C05440=1094.394,-80.468,-50.076,175.164,15.276,152.248
C05441=1094.401,-80.195,-50.087,175.166,15.277,152.248
C05442=1094.407,-79.945,-50.099,175.167,15.277,152.247
C05443=1094.413,-79.695,-50.109,175.169,15.278,152.247
C05444=1094.419,-79.446,-50.120,175.170,15.279,152.247
C05445=1094.425,-79.197,-50.131,175.172,15.279,152.247
C05446=1094.431,-78.946,-50.141,175.174,15.280,152.246
C05447=1094.437,-78.696,-50.152,175.175,15.280,152.246
C05448=1094.443,-78.447,-50.163,175.177,15.281,152.246
C05449=1094.448,-78.197,-50.174,175.179,15.282,152.246
C05450=1094.455,-77.947,-50.185,175.181,15.283,152.246
C05451=1094.461,-77.698,-50.195,175.182,15.284,152.245
C05452=1094.467,-77.449,-50.206,175.183,15.284,152.245
C05453=1094.473,-77.199,-50.217,175.185,15.285,152.245
C05454=1094.479,-76.948,-50.228,175.187,15.286,152.245
C05455=1094.484,-76.699,-50.238,175.189,15.286,152.244
C05456=1094.490,-76.449,-50.249,175.191,15.287,152.244
C05457=1094.497,-76.200,-50.260,175.192,15.288,152.244
C05458=1094.503,-75.950,-50.271,175.194,15.288,152.244
C05459=1094.509,-75.700,-50.282,175.195,15.289,152.244
C05460=1094.515,-75.451,-50.293,175.197,15.290,152.243
C05461=1094.521,-75.201,-50.304,175.199,15.291,152.243
C05462=1094.527,-74.951,-50.315,175.201,15.291,152.243
C05463=1094.532,-74.702,-50.326,175.203,15.292,152.243
C05464=1094.539,-74.453,-50.336,175.204,15.292,152.242
C05465=1094.545,-74.202,-50.347,175.205,15.293,152.242
C05466=1094.551,-73.953,-50.358,175.207,15.294,152.242
C05467=1094.557,-73.703,-50.369,175.209,15.295,152.242
C05468=1094.562,-73.453,-50.379,175.211,15.296,152.242
C05469=1094.568,-73.203,-50.390,175.213,15.297,152.241
C05470=1094.574,-72.954,-50.401,175.214,15.297,152.241
C05471=1094.580,-72.704,-50.412,175.215,15.298,152.241
C05472=1094.586,-72.455,-50.423,175.217,15.299,152.241
C05473=1094.592,-72.204,-50.434,175.219,15.299,152.241
C05474=1094.597,-71.955,-50.446,175.221,15.301,152.241
C05475=1094.603,-71.705,-50.457,175.223,15.301,152.240
C05476=1094.608,-71.456,-50.467,175.224,15.302,152.240
C05477=1094.615,-71.205,-50.479,175.225,15.302,152.240
C05478=1094.621,-70.956,-50.490,175.227,15.303,152.240
C05479=1094.627,-70.707,-50.501,175.229,15.304,152.239
C05480=1094.633,-70.457,-50.512,175.231,15.305,152.239
C05481=1094.639,-70.207,-50.523,175.233,15.306,152.239
C05482=1094.644,-69.958,-50.534,175.234,15.306,152.239
C05483=1094.650,-69.708,-50.545,175.236,15.308,152.239
C05484=1094.656,-69.458,-50.556,175.237,15.308,152.238
C05485=1094.662,-69.209,-50.567,175.239,15.308,152.238
C05486=1094.668,-68.959,-50.578,175.241,15.310,152.238
C05487=1094.674,-68.709,-50.589,175.242,15.310,152.238
C05488=1094.680,-68.460,-50.600,175.244,15.311,152.238
C05489=1094.685,-68.210,-50.612,175.246,15.312,152.237
C05490=1094.691,-67.960,-50.623,175.248,15.313,152.237
C05491=1094.697,-67.710,-50.634,175.250,15.314,152.237
C05492=1094.703,-67.461,-50.645,175.250,15.314,152.237
C05493=1094.709,-67.211,-50.657,175.252,15.315,152.237
C05494=1094.715,-66.962,-50.667,175.254,15.316,152.236
C05495=1094.721,-66.712,-50.678,175.256,15.317,152.236
C05496=1094.727,-66.462,-50.690,175.258,15.317,152.236
C05497=1094.733,-66.212,-50.700,175.260,15.318,152.236
C05498=1094.739,-65.963,-50.711,175.261,15.319,152.236
C05499=1094.745,-65.713,-50.724,175.263,15.320,152.235
C05500=1094.750,-65.464,-50.735,175.264,15.321,152.235
C05501=1094.757,-65.213,-50.746,175.266,15.321,152.235
C05502=1094.763,-64.943,-50.758,175.268,15.322,152.235
C05503=1094.769,-64.674,-50.769,175.270,15.323,152.235
C05504=1094.776,-64.404,-50.782,175.272,15.324,152.234
C05505=1094.782,-64.134,-50.794,175.274,15.325,152.234
C05506=1094.788,-63.884,-50.806,175.275,15.325,152.234
C05507=1094.794,-63.634,-50.816,175.277,15.326,152.234
C05508=1094.801,-63.385,-50.828,175.278,15.327,152.234
C05509=1094.806,-63.135,-50.839,175.280,15.328,152.233
C05510=1094.811,-62.885,-50.851,175.282,15.329,152.233
C05511=1094.818,-62.635,-50.862,175.284,15.330,152.233
C05512=1094.824,-62.386,-50.874,175.286,15.330,152.233
C05513=1094.830,-62.136,-50.885,175.287,15.332,152.233
C05514=1094.836,-61.887,-50.896,175.289,15.332,152.232
C05515=1094.842,-61.636,-50.907,175.291,15.333,152.232
C05516=1094.847,-61.387,-50.919,175.292,15.334,152.232
C05517=1094.853,-61.138,-50.930,175.294,15.334,152.232
C05518=1094.860,-60.888,-50.941,175.295,15.335,152.232
C05519=1094.866,-60.639,-50.953,175.297,15.336,152.231
C05520=1094.872,-60.389,-50.964,175.299,15.337,152.231
C05521=1094.878,-60.139,-50.975,175.301,15.338,152.231
C05522=1094.884,-59.889,-50.988,175.303,15.339,152.231
C05523=1094.889,-59.640,-50.998,175.304,15.339,152.230
C05524=1094.896,-59.390,-51.010,175.306,15.341,152.230
C05525=1094.902,-59.141,-51.021,175.308,15.341,152.230
C05526=1094.908,-58.890,-51.032,175.310,15.342,152.230
C05527=1094.913,-58.641,-51.044,175.311,15.343,152.230
C05528=1094.919,-58.392,-51.056,175.312,15.343,152.229
C05529=1094.925,-58.142,-51.067,175.314,15.344,152.229
C05530=1094.931,-57.892,-51.078,175.316,15.345,152.229
C05531=1094.937,-57.642,-51.090,175.318,15.346,152.229
C05532=1094.943,-57.393,-51.101,175.320,15.346,152.229
C05533=1094.949,-57.143,-51.113,175.321,15.348,152.228
C05534=1094.955,-56.894,-51.124,175.323,15.348,152.228
C05535=1094.962,-56.643,-51.135,175.325,15.349,152.228
C05536=1094.967,-56.394,-51.147,175.327,15.350,152.228
C05537=1094.973,-56.144,-51.159,175.329,15.351,152.228
C05538=1094.980,-55.895,-51.171,175.330,15.352,152.227
C05539=1094.986,-55.645,-51.181,175.332,15.353,152.227
C05540=1094.991,-55.395,-51.194,175.334,15.354,152.227
C05541=1094.997,-55.146,-51.205,175.336,15.354,152.227
C05542=1095.004,-54.896,-51.217,175.337,15.355,152.227
C05543=1095.010,-54.647,-51.228,175.339,15.355,152.226
C05544=1095.015,-54.397,-51.240,175.340,15.356,152.226
C05545=1095.021,-54.147,-51.251,175.342,15.357,152.226
C05546=1095.028,-53.898,-51.263,175.344,15.358,152.226
C05547=1095.033,-53.648,-51.275,175.346,15.359,152.225
C05548=1095.040,-53.398,-51.287,175.347,15.360,152.225
C05549=1095.046,-53.148,-51.298,175.349,15.361,152.225
C05550=1095.052,-52.899,-51.309,175.351,15.361,152.225
C05551=1095.058,-52.649,-51.321,175.353,15.363,152.225
C05552=1095.064,-52.400,-51.333,175.355,15.363,152.224
C05553=1095.070,-52.150,-51.344,175.356,15.364,152.224
C05554=1095.076,-51.901,-51.356,175.358,15.365,152.224
C05555=1095.082,-51.650,-51.367,175.360,15.366,152.224
C05556=1095.088,-51.401,-51.379,175.362,15.367,152.224
C05557=1095.094,-51.151,-51.390,175.363,15.368,152.223
C05558=1095.100,-50.901,-51.403,175.365,15.368,152.223
C05559=1095.106,-50.652,-51.414,175.367,15.370,152.223
C05560=1095.112,-50.402,-51.426,175.369,15.370,152.223
C05561=1095.118,-50.153,-51.438,175.371,15.371,152.223
C05562=1095.124,-49.903,-51.449,175.371,15.372,152.223
C05563=1095.129,-49.654,-51.461,175.373,15.372,152.222
C05564=1095.136,-49.404,-51.473,175.375,15.373,152.222
C05565=1095.141,-49.154,-51.485,175.377,15.374,152.222
C05566=1095.147,-48.885,-51.497,175.379,15.376,152.222
C05567=1095.153,-48.616,-51.511,175.381,15.377,152.222
C05568=1095.160,-48.347,-51.523,175.383,15.377,152.221
C05569=1095.166,-48.080,-51.536,175.385,15.378,152.221
C05570=1095.172,-47.829,-51.548,175.386,15.379,152.221
C05571=1095.178,-47.580,-51.559,175.388,15.380,152.221
C05572=1095.184,-47.330,-51.572,175.390,15.381,152.221
C05573=1095.190,-47.080,-51.583,175.392,15.382,152.220
C05574=1095.195,-46.831,-51.595,175.393,15.383,152.220
C05575=1095.202,-46.581,-51.607,175.395,15.384,152.220
C05576=1095.207,-46.332,-51.619,175.397,15.385,152.220
C05577=1095.214,-46.082,-51.631,175.399,15.386,152.220
C05578=1095.219,-45.833,-51.643,175.400,15.387,152.219
C05579=1095.225,-45.583,-51.655,175.402,15.387,152.219
C05580=1095.231,-45.333,-51.667,175.404,15.388,152.219
C05581=1095.237,-45.084,-51.679,175.406,15.389,152.219
C05582=1095.243,-44.834,-51.691,175.408,15.390,152.219
C05583=1095.248,-44.584,-51.702,175.409,15.391,152.218
C05584=1095.255,-44.335,-51.714,175.411,15.392,152.218
C05585=1095.261,-44.085,-51.727,175.413,15.393,152.218
C05586=1095.266,-43.836,-51.739,175.415,15.394,152.218
C05587=1095.272,-43.585,-51.750,175.416,15.394,152.218
C05588=1095.278,-43.335,-51.763,175.418,15.396,152.217
C05589=1095.284,-43.087,-51.774,175.420,15.396,152.217
C05590=1095.290,-42.837,-51.787,175.421,15.398,152.217
C05591=1095.295,-42.587,-51.798,175.423,15.398,152.217
C05592=1095.302,-42.337,-51.810,175.425,15.399,152.217
C05593=1095.308,-42.087,-51.823,175.427,15.400,152.216
C05594=1095.313,-41.838,-51.835,175.429,15.401,152.216
C05595=1095.320,-41.589,-51.847,175.430,15.402,152.216
C05596=1095.326,-41.339,-51.860,175.432,15.403,152.216
C05597=1095.331,-41.089,-51.871,175.434,15.404,152.216
C05598=1095.337,-40.839,-51.883,175.436,15.405,152.216
C05599=1095.343,-40.590,-51.896,175.438,15.405,152.215
C05600=1095.349,-40.341,-51.907,175.439,15.406,152.215
C05601=1095.355,-40.091,-51.920,175.441,15.407,152.215
C05602=1095.361,-39.841,-51.932,175.443,15.408,152.215
C05603=1095.367,-39.591,-51.943,175.445,15.409,152.215
C05604=1095.373,-39.342,-51.956,175.446,15.410,152.214
C05605=1095.379,-39.092,-51.968,175.448,15.411,152.214
C05606=1095.385,-38.842,-51.980,175.450,15.412,152.214
C05607=1095.391,-38.593,-51.992,175.451,15.413,152.214
C05608=1095.397,-38.343,-52.005,175.453,15.414,152.214
C05609=1095.402,-38.094,-52.017,175.455,15.415,152.213
C05610=1095.409,-37.844,-52.029,175.457,15.415,152.213
C05611=1095.414,-37.594,-52.042,175.458,15.417,152.213
C05612=1095.420,-37.345,-52.054,175.460,15.417,152.213
C05613=1095.425,-37.095,-52.066,175.462,15.418,152.213
C05614=1095.431,-36.845,-52.078,175.464,15.419,152.212
C05615=1095.437,-36.596,-52.090,175.466,15.420,152.212
C05616=1095.443,-36.346,-52.102,175.467,15.421,152.212
C05617=1095.449,-36.096,-52.115,175.469,15.422,152.212
C05618=1095.454,-35.847,-52.127,175.471,15.424,152.212
C05619=1095.460,-35.597,-52.140,175.473,15.424,152.211
C05620=1095.467,-35.348,-52.152,175.475,15.425,152.211
C05621=1095.473,-35.098,-52.164,175.477,15.426,152.211
C05622=1095.478,-34.848,-52.176,175.478,15.427,152.211
C05623=1095.484,-34.599,-52.189,175.480,15.428,152.211
C05624=1095.490,-34.349,-52.202,175.482,15.429,152.211
C05625=1095.495,-34.100,-52.214,175.484,15.430,152.210
C05626=1095.501,-33.850,-52.226,175.486,15.431,152.210
C05627=1095.508,-33.600,-52.238,175.487,15.432,152.210
C05628=1095.514,-33.350,-52.251,175.489,15.433,152.210
C05629=1095.519,-33.101,-52.263,175.491,15.434,152.210
C05630=1095.526,-32.832,-52.276,175.493,15.434,152.209
C05631=1095.532,-32.564,-52.290,175.494,15.436,152.209
C05632=1095.538,-32.296,-52.304,175.497,15.437,152.209
C05633=1095.545,-32.028,-52.317,175.499,15.438,152.209
C05634=1095.550,-31.769,-52.330,175.500,15.439,152.209
C05635=1095.557,-31.512,-52.342,175.502,15.439,152.208
C05636=1095.563,-31.253,-52.355,175.504,15.441,152.208
C05637=1095.569,-30.996,-52.369,175.506,15.441,152.208
C05638=1095.575,-30.746,-52.381,175.507,15.443,152.208
C05639=1095.581,-30.497,-52.393,175.510,15.444,152.208
C05640=1095.587,-30.247,-52.406,175.512,15.445,152.207
C05641=1095.593,-29.997,-52.418,175.513,15.446,152.207
C05642=1095.598,-29.747,-52.431,175.515,15.446,152.207
C05643=1095.604,-29.498,-52.443,175.517,15.448,152.207
C05644=1095.610,-29.249,-52.456,175.519,15.448,152.207
C05645=1095.616,-28.999,-52.469,175.521,15.449,152.206
C05646=1095.622,-28.749,-52.481,175.522,15.450,152.206
C05647=1095.628,-28.499,-52.494,175.524,15.451,152.206
C05648=1095.633,-28.250,-52.506,175.526,15.452,152.206
C05649=1095.640,-28.001,-52.519,175.528,15.453,152.206
C05650=1095.646,-27.751,-52.531,175.529,15.454,152.206
C05651=1095.652,-27.501,-52.544,175.531,15.455,152.205
C05652=1095.658,-27.251,-52.556,175.533,15.455,152.205
C05653=1095.664,-27.002,-52.569,175.535,15.457,152.205
C05654=1095.669,-26.753,-52.582,175.537,15.458,152.205
C05655=1095.675,-26.503,-52.594,175.539,15.459,152.205
C05656=1095.681,-26.253,-52.607,175.541,15.460,152.204
C05657=1095.686,-26.003,-52.620,175.542,15.461,152.204
C05658=1095.692,-25.754,-52.633,175.544,15.462,152.204
C05659=1095.698,-25.505,-52.646,175.546,15.463,152.204
C05660=1095.704,-25.255,-52.658,175.548,15.464,152.204
C05661=1095.709,-25.005,-52.671,175.550,15.464,152.203
C05662=1095.716,-24.756,-52.684,175.551,15.465,152.203
C05663=1095.722,-24.506,-52.696,175.553,15.466,152.203
C05664=1095.727,-24.256,-52.709,175.555,15.468,152.203
C05665=1095.733,-24.007,-52.721,175.557,15.469,152.203
C05666=1095.739,-23.757,-52.734,175.559,15.470,152.202
C05667=1095.744,-23.507,-52.748,175.561,15.471,152.202
C05668=1095.750,-23.257,-52.760,175.562,15.472,152.202
C05669=1095.756,-23.008,-52.773,175.564,15.472,152.202
C05670=1095.762,-22.759,-52.786,175.566,15.474,152.202
C05671=1095.768,-22.509,-52.798,175.568,15.474,152.201
C05672=1095.774,-22.260,-52.811,175.570,15.475,152.201
C05673=1095.780,-22.010,-52.824,175.572,15.477,152.201
C05674=1095.786,-21.760,-52.837,175.574,15.477,152.201
C05675=1095.791,-21.510,-52.850,175.575,15.479,152.201
C05676=1095.796,-21.261,-52.863,175.577,15.479,152.200
C05677=1095.803,-21.012,-52.876,175.579,15.481,152.200
C05678=1095.808,-20.762,-52.888,175.581,15.481,152.200
C05679=1095.814,-20.512,-52.901,175.583,15.482,152.200
C05680=1095.821,-20.263,-52.914,175.584,15.483,152.200
C05681=1095.826,-20.013,-52.927,175.586,15.484,152.200
C05682=1095.832,-19.763,-52.941,175.588,15.486,152.199
C05683=1095.838,-19.514,-52.953,175.590,15.486,152.199
C05684=1095.844,-19.264,-52.966,175.592,15.488,152.199
C05685=1095.850,-19.014,-52.979,175.594,15.488,152.199
C05686=1095.855,-18.765,-52.991,175.596,15.489,152.199
C05687=1095.861,-18.516,-53.005,175.597,15.490,152.198
C05688=1095.867,-18.266,-53.018,175.599,15.491,152.198
C05689=1095.873,-18.016,-53.031,175.601,15.492,152.198
C05690=1095.879,-17.767,-53.043,175.603,15.493,152.198
C05691=1095.885,-17.517,-53.057,175.605,15.494,152.197
C05692=1095.890,-17.267,-53.070,175.607,15.495,152.197
C05693=1095.896,-17.018,-53.083,175.609,15.496,152.197
C05694=1095.902,-16.757,-53.097,175.610,15.497,152.197
C05695=1095.909,-16.496,-53.111,175.612,15.498,152.197
C05696=1095.915,-16.235,-53.124,175.614,15.499,152.197
C05697=1095.921,-15.975,-53.138,175.617,15.500,152.196
C05698=1095.927,-15.725,-53.150,175.618,15.501,152.196
C05699=1095.933,-15.476,-53.164,175.620,15.502,152.196
C05700=1095.939,-15.226,-53.176,175.622,15.503,152.196
C05701=1095.944,-14.976,-53.190,175.624,15.504,152.196
C05702=1095.950,-14.726,-53.203,175.625,15.505,152.195
C05703=1095.956,-14.477,-53.216,175.628,15.506,152.195
C05704=1095.961,-14.227,-53.229,175.630,15.507,152.195
C05705=1095.968,-13.977,-53.242,175.631,15.508,152.195
C05706=1095.974,-13.728,-53.256,175.633,15.509,152.195
C05707=1095.979,-13.478,-53.269,175.635,15.510,152.194
C05708=1095.985,-13.229,-53.282,175.637,15.511,152.194
C05709=1095.990,-12.979,-53.295,175.638,15.512,152.194
C05710=1095.997,-12.729,-53.308,175.641,15.513,152.194
C05711=1096.003,-12.480,-53.322,175.643,15.514,152.194
C05712=1096.008,-12.230,-53.335,175.645,15.515,152.193
C05713=1096.014,-11.981,-53.348,175.646,15.516,152.193
C05714=1096.019,-11.732,-53.362,175.648,15.517,152.193
C05715=1096.025,-11.482,-53.374,175.650,15.518,152.193
C05716=1096.031,-11.233,-53.387,175.652,15.519,152.193
C05717=1096.037,-10.983,-53.401,175.654,15.520,152.192
C05718=1096.043,-10.733,-53.414,175.656,15.521,152.192
C05719=1096.048,-10.484,-53.428,175.658,15.522,152.192
C05720=1096.054,-10.234,-53.441,175.660,15.523,152.192
C05721=1096.059,-9.984,-53.454,175.661,15.524,152.192
C05722=1096.066,-9.735,-53.467,175.663,15.525,152.191
C05723=1096.072,-9.486,-53.481,175.666,15.526,152.191
C05724=1096.077,-9.236,-53.495,175.667,15.527,152.191
C05725=1096.083,-8.986,-53.507,175.669,15.528,152.191
C05726=1096.089,-8.737,-53.521,175.671,15.528,152.191
C05727=1096.095,-8.487,-53.534,175.673,15.530,152.190
C05728=1096.100,-8.238,-53.548,175.675,15.530,152.190
C05729=1096.107,-7.987,-53.561,175.677,15.532,152.190
C05730=1096.112,-7.738,-53.575,175.679,15.533,152.190
C05731=1096.119,-7.488,-53.588,175.681,15.534,152.190
C05732=1096.124,-7.239,-53.602,175.682,15.535,152.189
C05733=1096.130,-6.989,-53.615,175.684,15.535,152.189
C05734=1096.136,-6.739,-53.628,175.686,15.536,152.189
C05735=1096.142,-6.490,-53.642,175.688,15.538,152.189
C05736=1096.147,-6.240,-53.656,175.690,15.539,152.189
C05737=1096.153,-5.991,-53.669,175.692,15.539,152.188
C05738=1096.159,-5.742,-53.683,175.694,15.541,152.188
C05739=1096.165,-5.492,-53.695,175.696,15.541,152.188
C05740=1096.170,-5.242,-53.709,175.698,15.542,152.188
C05741=1096.176,-4.993,-53.722,175.700,15.544,152.188
C05742=1096.182,-4.743,-53.736,175.702,15.544,152.187
C05743=1096.188,-4.494,-53.750,175.704,15.545,152.187
C05744=1096.194,-4.244,-53.764,175.705,15.546,152.187
C05745=1096.200,-3.994,-53.777,175.707,15.547,152.187
C05746=1096.206,-3.745,-53.791,175.709,15.548,152.186
C05747=1096.212,-3.495,-53.803,175.711,15.549,152.186
C05748=1096.217,-3.245,-53.817,175.713,15.550,152.186
C05749=1096.224,-2.996,-53.831,175.715,15.551,152.186
C05750=1096.229,-2.747,-53.844,175.717,15.552,152.186
C05751=1096.234,-2.497,-53.858,175.719,15.553,152.185
C05752=1096.240,-2.247,-53.872,175.721,15.555,152.185
C05753=1096.246,-1.998,-53.885,175.723,15.555,152.185
C05754=1096.252,-1.749,-53.899,175.725,15.556,152.185
C05755=1096.257,-1.499,-53.913,175.726,15.557,152.185
C05756=1096.263,-1.250,-53.926,175.728,15.558,152.184
C05757=1096.269,-1.000,-53.940,175.731,15.560,152.184
C05758=1096.275,-0.729,-53.955,175.732,15.560,152.184
C05759=1096.281,-0.458,-53.970,175.734,15.561,152.184
C05760=1096.288,-0.188,-53.985,175.737,15.563,152.184
C05761=1096.294,0.084,-54.000,175.739,15.564,152.183
C05762=1096.299,0.333,-54.013,175.741,15.564,152.183
C05763=1096.305,0.583,-54.027,175.743,15.566,152.183
C05764=1096.312,0.833,-54.041,175.745,15.567,152.183
C05765=1096.317,1.082,-54.055,175.747,15.568,152.182
C05766=1096.322,1.332,-54.069,175.748,15.569,152.182
C05767=1096.328,1.581,-54.082,175.750,15.569,152.182
C05768=1096.333,1.831,-54.096,175.753,15.571,152.182
C05769=1096.340,2.080,-54.110,175.754,15.572,152.182
C05770=1096.345,2.329,-54.124,175.756,15.573,152.181
C05771=1096.351,2.579,-54.138,175.758,15.573,152.181
C05772=1096.357,2.829,-54.152,175.760,15.574,152.181
C05773=1096.363,3.078,-54.166,175.762,15.576,152.181
C05774=1096.369,3.328,-54.179,175.764,15.577,152.181
C05775=1096.374,3.577,-54.193,175.766,15.578,152.181
C05776=1096.380,3.827,-54.207,175.768,15.578,152.180
C05777=1096.385,4.077,-54.221,175.770,15.579,152.180
C05778=1096.391,4.326,-54.234,175.772,15.580,152.180
C05779=1096.398,4.576,-54.249,175.774,15.582,152.180
C05780=1096.403,4.825,-54.263,175.776,15.582,152.179
C05781=1096.409,5.075,-54.277,175.778,15.583,152.179
C05782=1096.414,5.324,-54.291,175.780,15.585,152.179
C05783=1096.420,5.574,-54.304,175.782,15.586,152.179
C05784=1096.426,5.824,-54.318,175.784,15.586,152.178
C05785=1096.432,6.073,-54.333,175.786,15.587,152.178
C05786=1096.438,6.322,-54.347,175.787,15.588,152.178
C05787=1096.443,6.572,-54.361,175.790,15.589,152.178
C05788=1096.449,6.821,-54.374,175.792,15.590,152.178
C05789=1096.455,7.071,-54.388,175.793,15.591,152.177
C05790=1096.461,7.320,-54.403,175.795,15.592,152.177
C05791=1096.467,7.570,-54.417,175.798,15.593,152.177
C05792=1096.472,7.820,-54.430,175.800,15.594,152.177
C05793=1096.478,8.070,-54.445,175.801,15.595,152.177
C05794=1096.484,8.319,-54.459,175.803,15.596,152.176
C05795=1096.489,8.568,-54.473,175.805,15.597,152.176
C05796=1096.496,8.818,-54.486,175.808,15.598,152.176
C05797=1096.502,9.068,-54.501,175.810,15.599,152.176
C05798=1096.508,9.317,-54.515,175.811,15.600,152.175
C05799=1096.513,9.566,-54.529,175.813,15.601,152.175
C05800=1096.519,9.816,-54.543,175.816,15.602,152.175
C05801=1096.525,10.066,-54.558,175.818,15.603,152.175
C05802=1096.530,10.315,-54.572,175.819,15.604,152.175
C05803=1096.536,10.565,-54.586,175.821,15.604,152.174
C05804=1096.542,10.814,-54.600,175.824,15.606,152.174
C05805=1096.548,11.064,-54.614,175.826,15.606,152.174
C05806=1096.554,11.313,-54.628,175.828,15.607,152.173
C05807=1096.560,11.562,-54.642,175.829,15.608,152.173
C05808=1096.566,11.813,-54.656,175.832,15.610,152.173
C05809=1096.571,12.062,-54.670,175.834,15.610,152.173
C05810=1096.577,12.311,-54.685,175.836,15.611,152.173
C05811=1096.583,12.561,-54.699,175.838,15.612,152.172
C05812=1096.589,12.810,-54.714,175.840,15.613,152.172
C05813=1096.594,13.060,-54.728,175.842,15.614,152.172
C05814=1096.600,13.310,-54.742,175.844,15.615,152.172
C05815=1096.606,13.559,-54.756,175.846,15.616,152.171
C05816=1096.612,13.809,-54.770,175.848,15.616,152.171
C05817=1096.618,14.058,-54.785,175.850,15.618,152.171
C05818=1096.624,14.308,-54.798,175.852,15.618,152.171
C05819=1096.629,14.557,-54.814,175.854,15.619,152.170
C05820=1096.635,14.807,-54.828,175.856,15.620,152.170
C05821=1096.641,15.056,-54.842,175.858,15.622,152.170
C05822=1096.648,15.329,-54.858,175.860,15.622,152.170
C05823=1096.654,15.601,-54.873,175.863,15.624,152.169
C05824=1096.660,15.874,-54.889,175.865,15.624,152.169
C05825=1096.667,16.147,-54.905,175.867,15.626,152.169
C05826=1096.672,16.397,-54.919,175.869,15.627,152.169
C05827=1096.678,16.646,-54.934,175.871,15.628,152.169
C05828=1096.684,16.896,-54.948,175.873,15.628,152.168
C05829=1096.689,17.145,-54.963,175.875,15.630,152.168
C05830=1096.695,17.395,-54.977,175.877,15.630,152.168
C05831=1096.701,17.645,-54.992,175.879,15.631,152.167
C05832=1096.706,17.894,-55.006,175.881,15.632,152.167
C05833=1096.712,18.143,-55.020,175.883,15.634,152.167
C05834=1096.718,18.393,-55.035,175.885,15.634,152.167
C05835=1096.724,18.642,-55.049,175.887,15.635,152.167
C05836=1096.730,18.891,-55.064,175.890,15.636,152.166
C05837=1096.735,19.142,-55.079,175.892,15.637,152.166
C05838=1096.741,19.391,-55.093,175.894,15.638,152.166
C05839=1096.747,19.641,-55.107,175.896,15.638,152.166
C05840=1096.753,19.890,-55.122,175.898,15.640,152.165
C05841=1096.759,20.139,-55.136,175.900,15.641,152.165
C05842=1096.765,20.389,-55.151,175.902,15.642,152.165
C05843=1096.770,20.639,-55.166,175.904,15.642,152.165
C05844=1096.776,20.888,-55.180,175.906,15.644,152.164
C05845=1096.782,21.138,-55.195,175.908,15.644,152.164
C05846=1096.787,21.387,-55.209,175.910,15.645,152.164
C05847=1096.793,21.637,-55.225,175.913,15.646,152.164
C05848=1096.799,21.886,-55.239,175.914,15.648,152.163
C05849=1096.804,22.135,-55.253,175.916,15.648,152.163
C05850=1096.811,22.385,-55.268,175.918,15.649,152.163
C05851=1096.815,22.635,-55.283,175.921,15.650,152.163
C05852=1096.822,22.885,-55.298,175.923,15.651,152.162
C05853=1096.828,23.134,-55.312,175.925,15.652,152.162
C05854=1096.832,23.383,-55.327,175.927,15.653,152.162
C05855=1096.839,23.633,-55.342,175.929,15.654,152.162
C05856=1096.844,23.882,-55.356,175.931,15.654,152.161
C05857=1096.851,24.132,-55.371,175.933,15.655,152.161
C05858=1096.856,24.382,-55.386,175.936,15.656,152.161
C05859=1096.862,24.631,-55.401,175.937,15.658,152.161
C05860=1096.868,24.880,-55.415,175.939,15.658,152.161
C05861=1096.873,25.130,-55.431,175.942,15.660,152.160
C05862=1096.879,25.379,-55.445,175.944,15.660,152.160
C05863=1096.885,25.629,-55.459,175.945,15.661,152.160
C05864=1096.890,25.879,-55.475,175.947,15.662,152.159
C05865=1096.896,26.128,-55.489,175.950,15.663,152.159
C05866=1096.902,26.377,-55.504,175.952,15.664,152.159
C05867=1096.908,26.627,-55.519,175.954,15.665,152.159
C05868=1096.914,26.876,-55.534,175.956,15.666,152.158
C05869=1096.919,27.126,-55.548,175.958,15.667,152.158
C05870=1096.925,27.376,-55.564,175.960,15.667,152.158
C05871=1096.931,27.625,-55.578,175.963,15.669,152.158
C05872=1096.937,27.874,-55.593,175.965,15.669,152.157
C05873=1096.942,28.124,-55.608,175.967,15.670,152.157
C05874=1096.949,28.373,-55.623,175.969,15.671,152.157
C05875=1096.954,28.622,-55.638,175.971,15.672,152.157
C05876=1096.960,28.872,-55.653,175.973,15.673,152.156
C05877=1096.966,29.122,-55.667,175.975,15.673,152.156
C05878=1096.971,29.372,-55.683,175.978,15.675,152.156
C05879=1096.977,29.621,-55.697,175.980,15.676,152.155
C05880=1096.983,29.871,-55.713,175.981,15.676,152.155
C05881=1096.988,30.120,-55.728,175.984,15.678,152.155
C05882=1096.994,30.370,-55.743,175.986,15.678,152.155
C05883=1097.000,30.619,-55.758,175.988,15.679,152.154
C05884=1097.005,30.868,-55.773,175.991,15.680,152.154
C05885=1097.011,31.117,-55.788,175.992,15.681,152.154
C05886=1097.017,31.392,-55.805,175.994,15.682,152.154
C05887=1097.023,31.666,-55.821,175.997,15.683,152.153
C05888=1097.030,31.940,-55.838,176.000,15.684,152.153
C05889=1097.037,32.214,-55.854,176.002,15.685,152.153
C05890=1097.042,32.464,-55.870,176.003,15.686,152.153
C05891=1097.048,32.713,-55.884,176.006,15.687,152.152
C05892=1097.054,32.963,-55.900,176.008,15.688,152.152
C05893=1097.059,33.212,-55.915,176.010,15.688,152.152
C05894=1097.065,33.462,-55.930,176.013,15.689,152.151
C05895=1097.070,33.711,-55.945,176.015,15.690,152.151
C05896=1097.076,33.961,-55.960,176.017,15.691,152.151
C05897=1097.082,34.211,-55.975,176.019,15.692,152.151
C05898=1097.088,34.460,-55.990,176.021,15.693,152.150
C05899=1097.094,34.709,-56.006,176.023,15.694,152.150
C05900=1097.100,34.958,-56.021,176.026,15.695,152.150
C05901=1097.105,35.208,-56.036,176.028,15.696,152.150
C05902=1097.111,35.457,-56.051,176.030,15.696,152.149
C05903=1097.117,35.707,-56.067,176.032,15.698,152.149
C05904=1097.122,35.957,-56.082,176.034,15.698,152.149
C05905=1097.128,36.206,-56.097,176.036,15.699,152.148
C05906=1097.134,36.456,-56.112,176.039,15.700,152.148
C05907=1097.140,36.704,-56.128,176.041,15.701,152.148
C05908=1097.145,36.954,-56.143,176.043,15.701,152.148
C05909=1097.151,37.204,-56.159,176.045,15.703,152.147
C05910=1097.157,37.453,-56.173,176.047,15.703,152.147
C05911=1097.163,37.703,-56.189,176.049,15.704,152.147
C05912=1097.169,37.952,-56.204,176.052,15.705,152.146
C05913=1097.174,38.201,-56.220,176.054,15.706,152.146
C05914=1097.180,38.451,-56.235,176.056,15.706,152.146
C05915=1097.185,38.701,-56.250,176.059,15.708,152.146
C05916=1097.191,38.950,-56.265,176.060,15.708,152.145
C05917=1097.197,39.200,-56.281,176.062,15.709,152.145
C05918=1097.202,39.449,-56.297,176.065,15.710,152.145
C05919=1097.209,39.699,-56.312,176.067,15.711,152.144
C05920=1097.214,39.948,-56.327,176.069,15.712,152.144
C05921=1097.220,40.197,-56.343,176.072,15.713,152.144
C05922=1097.225,40.447,-56.359,176.074,15.713,152.144
C05923=1097.231,40.696,-56.373,176.076,15.714,152.143
C05924=1097.237,40.945,-56.389,176.078,15.715,152.143
C05925=1097.243,41.195,-56.405,176.080,15.716,152.143
C05926=1097.248,41.445,-56.420,176.083,15.717,152.142
C05927=1097.253,41.695,-56.436,176.085,15.718,152.142
C05928=1097.260,41.943,-56.451,176.087,15.718,152.142
C05929=1097.265,42.193,-56.467,176.090,15.720,152.142
C05930=1097.271,42.442,-56.483,176.091,15.720,152.141
C05931=1097.276,42.692,-56.498,176.093,15.721,152.141
C05932=1097.283,42.941,-56.513,176.096,15.722,152.141
C05933=1097.288,43.191,-56.529,176.098,15.723,152.140
C05934=1097.294,43.441,-56.545,176.100,15.723,152.140
C05935=1097.299,43.690,-56.560,176.103,15.725,152.140
C05936=1097.305,43.939,-56.576,176.105,15.725,152.140
C05937=1097.311,44.189,-56.592,176.107,15.726,152.139
C05938=1097.316,44.438,-56.608,176.109,15.727,152.139
C05939=1097.322,44.688,-56.623,176.111,15.728,152.139
C05940=1097.327,44.937,-56.638,176.114,15.729,152.138
C05941=1097.334,45.186,-56.654,176.116,15.730,152.138
C05942=1097.339,45.436,-56.669,176.118,15.730,152.138
C05943=1097.345,45.685,-56.685,176.121,15.731,152.137
C05944=1097.350,45.935,-56.701,176.123,15.732,152.137
C05945=1097.356,46.184,-56.717,176.125,15.733,152.137
C05946=1097.361,46.433,-56.732,176.127,15.734,152.137
C05947=1097.367,46.683,-56.749,176.129,15.735,152.136
C05948=1097.373,46.933,-56.764,176.132,15.736,152.136
C05949=1097.378,47.181,-56.780,176.134,15.736,152.136
C05950=1097.384,47.456,-56.798,176.137,15.738,152.135
C05951=1097.390,47.730,-56.815,176.139,15.738,152.135
C05952=1097.397,48.005,-56.832,176.141,15.739,152.135
C05953=1097.403,48.279,-56.850,176.143,15.740,152.134
C05954=1097.408,48.528,-56.865,176.146,15.741,152.134
C05955=1097.414,48.778,-56.882,176.148,15.741,152.134
C05956=1097.420,49.028,-56.897,176.151,15.743,152.133
C05957=1097.426,49.277,-56.913,176.153,15.743,152.133
C05958=1097.431,49.526,-56.929,176.155,15.744,152.133
C05959=1097.437,49.776,-56.945,176.158,15.745,152.132
C05960=1097.442,50.025,-56.961,176.159,15.746,152.132
C05961=1097.448,50.275,-56.977,176.162,15.746,152.132
C05962=1097.453,50.524,-56.993,176.164,15.747,152.132
C05963=1097.459,50.773,-57.008,176.166,15.748,152.131
C05964=1097.465,51.023,-57.024,176.169,15.749,152.131
C05965=1097.471,51.272,-57.041,176.171,15.750,152.131
C05966=1097.476,51.521,-57.056,176.173,15.750,152.130
C05967=1097.482,51.771,-57.072,176.176,15.751,152.130
C05968=1097.488,52.020,-57.088,176.178,15.752,152.130
C05969=1097.494,52.270,-57.104,176.181,15.753,152.129
C05970=1097.500,52.519,-57.120,176.183,15.753,152.129
C05971=1097.505,52.768,-57.136,176.185,15.754,152.129
C05972=1097.511,53.018,-57.152,176.188,15.755,152.128
C05973=1097.517,53.267,-57.168,176.189,15.756,152.128
C05974=1097.522,53.517,-57.185,176.192,15.757,152.128
C05975=1097.528,53.766,-57.201,176.194,15.757,152.127
C05976=1097.533,54.016,-57.216,176.196,15.758,152.127
C05977=1097.539,54.265,-57.232,176.199,15.759,152.127
C05978=1097.545,54.514,-57.249,176.201,15.760,152.126
C05979=1097.551,54.764,-57.265,176.203,15.760,152.126
C05980=1097.556,55.014,-57.280,176.206,15.761,152.126
C05981=1097.562,55.263,-57.297,176.208,15.762,152.125
C05982=1097.568,55.512,-57.313,176.211,15.763,152.125
C05983=1097.573,55.761,-57.329,176.213,15.763,152.125
C05984=1097.579,56.011,-57.346,176.215,15.764,152.124
C05985=1097.584,56.261,-57.361,176.218,15.765,152.124
C05986=1097.590,56.510,-57.377,176.220,15.765,152.124
C05987=1097.596,56.759,-57.394,176.222,15.767,152.123
C05988=1097.602,57.009,-57.410,176.225,15.767,152.123
C05989=1097.608,57.258,-57.426,176.226,15.768,152.123
C05990=1097.614,57.507,-57.442,176.229,15.768,152.122
C05991=1097.619,57.756,-57.459,176.231,15.769,152.122
C05992=1097.624,58.006,-57.474,176.234,15.770,152.122
C05993=1097.630,58.256,-57.491,176.236,15.771,152.121
C05994=1097.636,58.505,-57.507,176.238,15.771,152.121
C05995=1097.642,58.754,-57.523,176.241,15.772,152.121
C05996=1097.648,59.004,-57.539,176.243,15.772,152.120
C05997=1097.653,59.253,-57.556,176.246,15.774,152.120
C05998=1097.659,59.503,-57.573,176.248,15.774,152.120
C05999=1097.665,59.752,-57.589,176.251,15.775,152.119
C06000=1097.671,60.001,-57.605,176.253,15.776,152.119
C06001=1097.677,60.251,-57.621,176.255,15.776,152.118
C06002=1097.683,60.500,-57.638,176.258,15.777,152.118
C06003=1097.688,60.750,-57.654,176.260,15.777,152.118
C06004=1097.694,60.999,-57.671,176.263,15.779,152.117
C06005=1097.700,61.249,-57.687,176.265,15.779,152.117
C06006=1097.706,61.498,-57.703,176.267,15.779,152.117
C06007=1097.711,61.748,-57.720,176.270,15.781,152.116
C06008=1097.717,61.997,-57.736,176.272,15.781,152.116
C06009=1097.723,62.246,-57.753,176.275,15.782,152.116
C06010=1097.729,62.496,-57.769,176.277,15.782,152.115
C06011=1097.735,62.745,-57.785,176.279,15.783,152.115
C06012=1097.740,62.995,-57.802,176.282,15.783,152.114
C06013=1097.746,63.244,-57.818,176.284,15.784,152.114
C06014=1097.753,63.517,-57.836,176.287,15.785,152.114
C06015=1097.759,63.792,-57.854,176.290,15.786,152.113
C06016=1097.765,64.066,-57.873,176.292,15.786,152.113
C06017=1097.772,64.340,-57.891,176.295,15.787,152.112
C06018=1097.777,64.590,-57.907,176.297,15.788,152.112
C06019=1097.783,64.839,-57.924,176.300,15.789,152.112
C06020=1097.789,65.088,-57.940,176.302,15.789,152.111
C06021=1097.794,65.338,-57.957,176.305,15.790,152.111
C06022=1097.801,65.587,-57.974,176.307,15.790,152.111
C06023=1097.806,65.836,-57.991,176.309,15.791,152.110
C06024=1097.812,66.086,-58.007,176.312,15.792,152.110
C06025=1097.818,66.335,-58.023,176.314,15.792,152.110
C06026=1097.823,66.585,-58.040,176.317,15.793,152.109
C06027=1097.829,66.834,-58.056,176.319,15.794,152.109
C06028=1097.835,67.083,-58.074,176.322,15.795,152.108
C06029=1097.840,67.332,-58.090,176.324,15.795,152.108
C06030=1097.846,67.582,-58.107,176.326,15.796,152.108
C06031=1097.852,67.831,-58.123,176.329,15.797,152.107
C06032=1097.857,68.081,-58.140,176.331,15.797,152.107
C06033=1097.863,68.330,-58.157,176.334,15.798,152.107
C06034=1097.868,68.579,-58.174,176.336,15.798,152.106
C06035=1097.874,68.829,-58.190,176.339,15.799,152.106
C06036=1097.880,69.078,-58.206,176.341,15.799,152.105
C06037=1097.886,69.327,-58.224,176.344,15.801,152.105
C06038=1097.892,69.576,-58.240,176.346,15.801,152.105
C06039=1097.897,69.826,-58.257,176.348,15.801,152.104
C06040=1097.902,70.075,-58.275,176.351,15.802,152.104
C06041=1097.908,70.325,-58.291,176.353,15.803,152.104
C06042=1097.914,70.574,-58.308,176.356,15.804,152.103
C06043=1097.920,70.823,-58.325,176.358,15.804,152.103
C06044=1097.925,71.073,-58.342,176.361,15.805,152.102
C06045=1097.931,71.322,-58.358,176.363,15.806,152.102
C06046=1097.937,71.571,-58.375,176.366,15.806,152.102
C06047=1097.942,71.821,-58.393,176.368,15.807,152.101
C06048=1097.948,72.071,-58.409,176.370,15.807,152.101
C06049=1097.954,72.320,-58.426,176.373,15.808,152.101
C06050=1097.960,72.569,-58.443,176.375,15.808,152.100
C06051=1097.965,72.819,-58.459,176.378,15.809,152.100
C06052=1097.970,73.068,-58.477,176.380,15.810,152.099
C06053=1097.976,73.317,-58.493,176.383,15.810,152.099
C06054=1097.982,73.566,-58.511,176.385,15.811,152.099
C06055=1097.987,73.816,-58.528,176.388,15.812,152.098
C06056=1097.993,74.065,-58.545,176.390,15.812,152.098
C06057=1097.999,74.315,-58.562,176.393,15.813,152.097
C06058=1098.004,74.565,-58.579,176.395,15.813,152.097
C06059=1098.011,74.813,-58.596,176.397,15.814,152.097
C06060=1098.016,75.063,-58.613,176.400,15.815,152.096
C06061=1098.021,75.312,-58.630,176.402,15.815,152.096
C06062=1098.027,75.561,-58.646,176.405,15.816,152.095
C06063=1098.033,75.810,-58.664,176.408,15.816,152.095
C06064=1098.038,76.060,-58.681,176.410,15.817,152.095
C06065=1098.045,76.309,-58.698,176.413,15.817,152.094
C06066=1098.050,76.559,-58.715,176.416,15.818,152.094
C06067=1098.056,76.808,-58.733,176.418,15.819,152.093
C06068=1098.062,77.057,-58.750,176.421,15.819,152.093
C06069=1098.067,77.307,-58.766,176.423,15.820,152.093
C06070=1098.073,77.556,-58.784,176.425,15.820,152.092
C06071=1098.079,77.806,-58.801,176.428,15.821,152.092
C06072=1098.085,78.055,-58.818,176.430,15.821,152.091
C06073=1098.090,78.304,-58.835,176.433,15.822,152.091
C06074=1098.096,78.553,-58.853,176.435,15.823,152.091
C06075=1098.101,78.802,-58.870,176.438,15.824,152.090
C06076=1098.108,79.052,-58.887,176.440,15.824,152.090
C06077=1098.113,79.302,-58.904,176.443,15.825,152.089
C06078=1098.119,79.575,-58.923,176.445,15.825,152.089
C06079=1098.125,79.849,-58.942,176.448,15.826,152.088
C06080=1098.131,80.123,-58.962,176.452,15.826,152.088
C06081=1098.137,80.397,-58.980,176.455,15.827,152.087
C06082=1098.143,80.646,-58.997,176.457,15.827,152.087
C06083=1098.149,80.896,-59.015,176.460,15.828,152.087
C06084=1098.154,81.146,-59.032,176.462,15.828,152.086
C06085=1098.160,81.395,-59.050,176.465,15.829,152.086
C06086=1098.165,81.644,-59.067,176.467,15.830,152.085
C06087=1098.170,81.893,-59.084,176.469,15.830,152.085
C06088=1098.177,82.143,-59.102,176.472,15.831,152.085
C06089=1098.183,82.392,-59.119,176.475,15.831,152.084
C06090=1098.188,82.641,-59.137,176.478,15.832,152.084
C06091=1098.193,82.891,-59.154,176.480,15.832,152.083
C06092=1098.200,83.140,-59.171,176.483,15.833,152.083
C06093=1098.205,83.389,-59.189,176.485,15.833,152.082
C06094=1098.211,83.638,-59.207,176.488,15.834,152.082
C06095=1098.216,83.888,-59.223,176.490,15.834,152.082
C06096=1098.222,84.138,-59.241,176.493,15.835,152.081
C06097=1098.227,84.387,-59.259,176.495,15.835,152.081
C06098=1098.233,84.636,-59.277,176.498,15.836,152.080
C06099=1098.239,84.885,-59.294,176.500,15.837,152.080
C06100=1098.245,85.135,-59.312,176.503,15.837,152.079
C06101=1098.250,85.384,-59.329,176.505,15.838,152.079
C06102=1098.255,85.633,-59.346,176.509,15.838,152.078
C06103=1098.261,85.883,-59.364,176.511,15.838,152.078
C06104=1098.268,86.132,-59.381,176.514,15.839,152.078
C06105=1098.273,86.381,-59.399,176.516,15.839,152.077
C06106=1098.279,86.630,-59.416,176.519,15.840,152.077
C06107=1098.285,86.880,-59.434,176.521,15.841,152.076
C06108=1098.290,87.129,-59.452,176.524,15.841,152.076
C06109=1098.296,87.378,-59.470,176.527,15.841,152.075
C06110=1098.302,87.628,-59.487,176.530,15.842,152.075
C06111=1098.307,87.877,-59.504,176.532,15.842,152.075
C06112=1098.313,88.126,-59.522,176.535,15.843,152.074
C06113=1098.319,88.376,-59.540,176.537,15.843,152.074
C06114=1098.324,88.625,-59.557,176.540,15.844,152.073
C06115=1098.331,88.875,-59.575,176.542,15.844,152.073
C06116=1098.336,89.124,-59.593,176.545,15.845,152.072
C06117=1098.341,89.373,-59.611,176.548,15.845,152.072
C06118=1098.347,89.623,-59.629,176.551,15.846,152.071
C06119=1098.352,89.872,-59.647,176.553,15.846,152.071
C06120=1098.358,90.121,-59.664,176.556,15.847,152.070
C06121=1098.364,90.371,-59.682,176.558,15.847,152.070
C06122=1098.370,90.620,-59.700,176.561,15.847,152.069
C06123=1098.376,90.869,-59.718,176.564,15.848,152.069
C06124=1098.382,91.118,-59.736,176.567,15.849,152.069
C06125=1098.387,91.367,-59.753,176.569,15.849,152.068
C06126=1098.393,91.617,-59.771,176.572,15.849,152.068
C06127=1098.398,91.866,-59.790,176.574,15.850,152.067
C06128=1098.404,92.115,-59.807,176.577,15.850,152.067
C06129=1098.410,92.365,-59.825,176.579,15.851,152.066
C06130=1098.415,92.614,-59.843,176.583,15.851,152.066
C06131=1098.421,92.863,-59.860,176.585,15.851,152.065
C06132=1098.426,93.113,-59.879,176.588,15.852,152.065
C06133=1098.432,93.362,-59.896,176.590,15.852,152.065
C06134=1098.438,93.611,-59.915,176.593,15.853,152.064
C06135=1098.444,93.860,-59.932,176.595,15.853,152.064
C06136=1098.448,94.109,-59.951,176.598,15.854,152.063
C06137=1098.454,94.359,-59.969,176.601,15.854,152.063
C06138=1098.460,94.608,-59.986,176.604,15.855,152.062
C06139=1098.466,94.857,-60.005,176.606,15.855,152.062
C06140=1098.471,95.107,-60.023,176.609,15.855,152.061
C06141=1098.477,95.356,-60.040,176.612,15.856,152.061
C06142=1098.483,95.630,-60.060,176.615,15.856,152.060
C06143=1098.489,95.904,-60.080,176.618,15.857,152.060
C06144=1098.496,96.177,-60.100,176.621,15.857,152.059
C06145=1098.502,96.451,-60.120,176.623,15.858,152.059
C06146=1098.508,96.701,-60.138,176.627,15.858,152.058
C06147=1098.513,96.950,-60.156,176.629,15.858,152.058
C06148=1098.519,97.200,-60.175,176.632,15.859,152.057
C06149=1098.524,97.449,-60.192,176.634,15.859,152.057
C06150=1098.530,97.698,-60.210,176.637,15.859,152.056
C06151=1098.536,97.948,-60.228,176.640,15.860,152.056
C06152=1098.542,98.197,-60.247,176.643,15.860,152.055
C06153=1098.547,98.446,-60.265,176.645,15.860,152.055
C06154=1098.553,98.696,-60.283,176.648,15.861,152.054
C06155=1098.558,98.944,-60.302,176.651,15.861,152.054
C06156=1098.565,99.194,-60.319,176.653,15.862,152.053
C06157=1098.570,99.443,-60.338,176.656,15.862,152.053
C06158=1098.576,99.693,-60.356,176.659,15.863,152.052
C06159=1098.581,99.942,-60.374,176.662,15.863,152.052
C06160=1098.588,100.191,-60.392,176.664,15.863,152.051
C06161=1098.592,100.440,-60.411,176.668,15.864,152.051
C06162=1098.599,100.689,-60.429,176.670,15.864,152.050
C06163=1098.604,100.938,-60.447,176.673,15.864,152.050
C06164=1098.610,101.188,-60.465,176.676,15.864,152.049
C06165=1098.616,101.438,-60.484,176.679,15.865,152.049
C06166=1098.621,101.687,-60.502,176.681,15.865,152.048
C06167=1098.627,101.936,-60.521,176.684,15.866,152.048
C06168=1098.632,102.185,-60.539,176.686,15.865,152.047
C06169=1098.639,102.434,-60.558,176.689,15.866,152.047
C06170=1098.643,102.684,-60.576,176.692,15.866,152.046
C06171=1098.650,102.933,-60.594,176.695,15.867,152.046
C06172=1098.655,103.182,-60.613,176.697,15.867,152.045
C06173=1098.661,103.431,-60.631,176.700,15.868,152.045
C06174=1098.666,103.681,-60.649,176.703,15.868,152.044
C06175=1098.672,103.930,-60.668,176.706,15.868,152.044
C06176=1098.677,104.179,-60.686,176.709,15.869,152.043
C06177=1098.683,104.428,-60.705,176.711,15.869,152.043
C06178=1098.689,104.677,-60.724,176.715,15.869,152.042
C06179=1098.694,104.927,-60.742,176.717,15.869,152.042
C06180=1098.700,105.176,-60.761,176.720,15.870,152.041
C06181=1098.705,105.426,-60.779,176.722,15.870,152.041
C06182=1098.712,105.675,-60.798,176.725,15.871,152.040
C06183=1098.717,105.923,-60.817,176.728,15.871,152.040
C06184=1098.723,106.173,-60.835,176.731,15.871,152.039
C06185=1098.728,106.422,-60.853,176.733,15.871,152.039
C06186=1098.733,106.672,-60.872,176.737,15.872,152.038
C06187=1098.740,106.921,-60.891,176.740,15.872,152.038
C06188=1098.745,107.170,-60.910,176.742,15.872,152.037
C06189=1098.751,107.420,-60.927,176.745,15.873,152.037
C06190=1098.757,107.669,-60.947,176.748,15.873,152.036
C06191=1098.762,107.918,-60.966,176.751,15.874,152.036
C06192=1098.768,108.167,-60.984,176.753,15.873,152.035
C06193=1098.773,108.416,-61.002,176.757,15.874,152.034
C06194=1098.779,108.665,-61.021,176.759,15.874,152.034
C06195=1098.785,108.915,-61.040,176.762,15.875,152.033
C06196=1098.790,109.164,-61.058,176.764,15.874,152.033
C06197=1098.796,109.413,-61.077,176.768,15.875,152.032
C06198=1098.802,109.663,-61.096,176.771,15.875,152.032
C06199=1098.808,109.911,-61.115,176.773,15.875,152.031
C06200=1098.813,110.161,-61.134,176.776,15.876,152.031
C06201=1098.819,110.411,-61.152,176.779,15.876,152.030
C06202=1098.825,110.659,-61.171,176.782,15.876,152.030
C06203=1098.830,110.908,-61.190,176.785,15.876,152.029
C06204=1098.836,111.158,-61.209,176.788,15.877,152.029
C06205=1098.842,111.407,-61.228,176.790,15.877,152.028
C06206=1098.848,111.681,-61.248,176.793,15.877,152.027
C06207=1098.854,111.955,-61.269,176.797,15.877,152.027
C06208=1098.861,112.229,-61.290,176.800,15.878,152.026
C06209=1098.867,112.503,-61.310,176.804,15.878,152.025
C06210=1098.873,112.752,-61.330,176.806,15.878,152.025
C06211=1098.878,113.001,-61.349,176.809,15.879,152.024
C06212=1098.883,113.251,-61.367,176.811,15.878,152.024
C06213=1098.889,113.501,-61.386,176.815,15.879,152.023
C06214=1098.895,113.750,-61.405,176.817,15.879,152.023
C06215=1098.900,113.998,-61.424,176.820,15.879,152.022
C06216=1098.906,114.248,-61.443,176.824,15.879,152.022
C06217=1098.912,114.497,-61.462,176.826,15.880,152.021
C06218=1098.917,114.746,-61.481,176.829,15.880,152.021
C06219=1098.922,114.995,-61.500,176.832,15.880,152.020
C06220=1098.929,115.245,-61.519,176.835,15.880,152.019
C06221=1098.935,115.494,-61.538,176.837,15.880,152.019
C06222=1098.940,115.743,-61.557,176.841,15.881,152.018
C06223=1098.945,115.992,-61.576,176.843,15.881,152.018
C06224=1098.951,116.242,-61.596,176.846,15.881,152.017
C06225=1098.956,116.490,-61.615,176.849,15.882,152.017
C06226=1098.962,116.740,-61.634,176.852,15.882,152.016
C06227=1098.967,116.989,-61.653,176.855,15.882,152.016
C06228=1098.973,117.239,-61.672,176.858,15.882,152.015
C06229=1098.978,117.487,-61.691,176.861,15.882,152.014
C06230=1098.984,117.737,-61.710,176.864,15.883,152.014
C06231=1098.990,117.986,-61.730,176.866,15.883,152.013
C06232=1098.995,118.235,-61.749,176.870,15.883,152.013
C06233=1099.000,118.484,-61.768,176.872,15.883,152.012
C06234=1099.006,118.733,-61.788,176.875,15.884,152.012
C06235=1099.012,118.983,-61.807,176.878,15.883,152.011
C06236=1099.018,119.232,-61.826,176.881,15.884,152.011
C06237=1099.023,119.481,-61.845,176.884,15.884,152.010
C06238=1099.029,119.730,-61.864,176.887,15.884,152.009
C06239=1099.034,119.980,-61.884,176.890,15.885,152.009
C06240=1099.040,120.229,-61.903,176.893,15.884,152.008
C06241=1099.046,120.478,-61.923,176.896,15.885,152.008
C06242=1099.051,120.727,-61.942,176.898,15.885,152.007
C06243=1099.057,120.976,-61.961,176.902,15.885,152.007
C06244=1099.062,121.225,-61.980,176.905,15.886,152.006
C06245=1099.068,121.475,-61.999,176.907,15.885,152.005
C06246=1099.074,121.724,-62.019,176.911,15.886,152.005
C06247=1099.079,121.972,-62.038,176.913,15.886,152.004
C06248=1099.085,122.222,-62.057,176.917,15.886,152.004
C06249=1099.091,122.471,-62.077,176.920,15.886,152.003
C06250=1099.097,122.720,-62.097,176.922,15.886,152.002
C06251=1099.102,122.970,-62.116,176.926,15.886,152.002
C06252=1099.107,123.219,-62.136,176.928,15.886,152.001
C06253=1099.113,123.468,-62.156,176.931,15.887,152.001
C06254=1099.118,123.717,-62.175,176.934,15.886,152.000
C06255=1099.124,123.966,-62.194,176.937,15.887,152.000
C06256=1099.130,124.215,-62.214,176.940,15.887,151.999
C06257=1099.136,124.465,-62.233,176.943,15.887,151.998
C06258=1099.141,124.714,-62.252,176.946,15.887,151.998
C06259=1099.147,124.963,-62.272,176.949,15.887,151.997
C06260=1099.153,125.212,-62.291,176.952,15.887,151.997
C06261=1099.159,125.462,-62.311,176.956,15.888,151.996
C06262=1099.164,125.711,-62.331,176.958,15.887,151.995
C06263=1099.170,125.960,-62.351,176.962,15.888,151.995
C06264=1099.175,126.208,-62.370,176.964,15.887,151.994
C06265=1099.181,126.458,-62.389,176.967,15.888,151.994
C06266=1099.186,126.707,-62.409,176.970,15.888,151.993
C06267=1099.192,126.956,-62.429,176.973,15.888,151.992
C06268=1099.198,127.205,-62.448,176.977,15.888,151.992
C06269=1099.204,127.454,-62.468,176.979,15.888,151.991
C06270=1099.210,127.729,-62.489,176.983,15.888,151.990
C06271=1099.217,128.003,-62.512,176.986,15.888,151.990
C06272=1099.222,128.277,-62.533,176.989,15.888,151.989
C06273=1099.229,128.550,-62.554,176.993,15.888,151.988
C06274=1099.234,128.800,-62.574,176.996,15.888,151.988
C06275=1099.240,129.049,-62.594,176.999,15.889,151.987
C06276=1099.246,129.298,-62.613,177.002,15.888,151.986
C06277=1099.252,129.547,-62.633,177.005,15.888,151.986
C06278=1099.258,129.797,-62.653,177.008,15.889,151.985
C06279=1099.263,130.046,-62.673,177.011,15.888,151.985
C06280=1099.269,130.294,-62.693,177.014,15.889,151.984
C06281=1099.274,130.544,-62.712,177.017,15.888,151.983
C06282=1099.280,130.793,-62.732,177.020,15.888,151.983
C06283=1099.286,131.042,-62.752,177.023,15.889,151.982
C06284=1099.291,131.291,-62.772,177.026,15.888,151.981
C06285=1099.297,131.540,-62.792,177.030,15.889,151.981
C06286=1099.303,131.790,-62.811,177.032,15.888,151.980
C06287=1099.309,132.038,-62.831,177.036,15.889,151.979
C06288=1099.314,132.287,-62.852,177.039,15.889,151.979
C06289=1099.320,132.537,-62.871,177.042,15.888,151.978
C06290=1099.326,132.786,-62.891,177.045,15.889,151.978
C06291=1099.331,133.035,-62.912,177.048,15.888,151.977
C06292=1099.337,133.284,-62.931,177.051,15.889,151.976
C06293=1099.342,133.533,-62.951,177.054,15.889,151.976
C06294=1099.348,133.782,-62.971,177.057,15.888,151.975
C06295=1099.355,134.032,-62.992,177.060,15.889,151.974
C06296=1099.360,134.281,-63.012,177.063,15.888,151.974
C06297=1099.366,134.530,-63.032,177.066,15.889,151.973
C06298=1099.371,134.779,-63.052,177.070,15.889,151.973
C06299=1099.377,135.028,-63.072,177.072,15.889,151.972
C06300=1099.382,135.278,-63.092,177.076,15.889,151.971
C06301=1099.388,135.527,-63.112,177.079,15.889,151.970
C06302=1099.394,135.776,-63.132,177.082,15.889,151.970
C06303=1099.399,136.025,-63.152,177.085,15.889,151.969
C06304=1099.405,136.273,-63.172,177.088,15.889,151.969
C06305=1099.410,136.523,-63.192,177.091,15.889,151.968
C06306=1099.416,136.772,-63.212,177.094,15.889,151.967
C06307=1099.421,137.021,-63.233,177.097,15.889,151.967
C06308=1099.427,137.270,-63.253,177.101,15.889,151.966
C06309=1099.433,137.520,-63.274,177.103,15.888,151.965
C06310=1099.439,137.769,-63.293,177.107,15.889,151.965
C06311=1099.445,138.018,-63.314,177.110,15.889,151.964
C06312=1099.450,138.267,-63.333,177.113,15.888,151.963
C06313=1099.455,138.516,-63.354,177.116,15.889,151.963
C06314=1099.461,138.765,-63.374,177.120,15.889,151.962
C06315=1099.467,139.014,-63.394,177.122,15.888,151.961
C06316=1099.473,139.263,-63.414,177.126,15.888,151.961
C06317=1099.479,139.513,-63.435,177.128,15.888,151.960
C06318=1099.485,139.762,-63.455,177.132,15.888,151.959
C06319=1099.490,140.011,-63.476,177.135,15.888,151.959
C06320=1099.495,140.260,-63.496,177.138,15.888,151.958
C06321=1099.501,140.509,-63.516,177.141,15.888,151.957
C06322=1099.506,140.758,-63.537,177.145,15.889,151.957
C06323=1099.512,141.007,-63.557,177.147,15.888,151.956
C06324=1099.518,141.257,-63.578,177.151,15.888,151.955
C06325=1099.523,141.506,-63.598,177.154,15.888,151.955
C06326=1099.529,141.754,-63.618,177.157,15.888,151.954
C06327=1099.535,142.004,-63.639,177.160,15.888,151.953
C06328=1099.540,142.253,-63.659,177.163,15.888,151.953
C06329=1099.546,142.502,-63.679,177.167,15.888,151.952
C06330=1099.551,142.751,-63.700,177.170,15.888,151.951
C06331=1099.557,143.000,-63.721,177.173,15.888,151.951
C06332=1099.563,143.249,-63.741,177.176,15.888,151.950
C06333=1099.569,143.498,-63.762,177.180,15.888,151.949
C06334=1099.574,143.772,-63.785,177.182,15.887,151.949
C06335=1099.581,144.046,-63.807,177.186,15.887,151.948
C06336=1099.587,144.320,-63.829,177.190,15.887,151.947
C06337=1099.593,144.594,-63.853,177.193,15.887,151.946
C06338=1099.599,144.842,-63.873,177.197,15.887,151.946
C06339=1099.604,145.092,-63.893,177.199,15.887,151.945
C06340=1099.610,145.341,-63.914,177.203,15.887,151.944
C06341=1099.616,145.590,-63.934,177.207,15.887,151.943
C06342=1099.622,145.839,-63.956,177.209,15.887,151.943
C06343=1099.627,146.088,-63.976,177.213,15.887,151.942
C06344=1099.632,146.337,-63.997,177.216,15.887,151.941
C06345=1099.639,146.586,-64.017,177.219,15.886,151.941
C06346=1099.644,146.836,-64.038,177.222,15.886,151.940
C06347=1099.650,147.084,-64.059,177.226,15.887,151.939
C06348=1099.655,147.333,-64.079,177.229,15.886,151.939
C06349=1099.662,147.583,-64.100,177.232,15.886,151.938
C06350=1099.667,147.831,-64.121,177.235,15.885,151.937
C06351=1099.672,148.080,-64.142,177.238,15.885,151.937
C06352=1099.678,148.330,-64.162,177.242,15.885,151.936
C06353=1099.684,148.579,-64.184,177.244,15.885,151.935
C06354=1099.689,148.828,-64.204,177.248,15.885,151.934
C06355=1099.695,149.077,-64.224,177.252,15.885,151.934
C06356=1099.701,149.326,-64.246,177.254,15.885,151.933
C06357=1099.706,149.575,-64.266,177.258,15.885,151.932
C06358=1099.712,149.824,-64.287,177.261,15.885,151.932
C06359=1099.718,150.073,-64.309,177.264,15.884,151.931
C06360=1099.723,150.322,-64.329,177.268,15.885,151.930
C06361=1099.729,150.571,-64.350,177.271,15.885,151.930
C06362=1099.735,150.821,-64.371,177.274,15.884,151.929
C06363=1099.740,151.070,-64.392,177.277,15.884,151.928
C06364=1099.745,151.318,-64.413,177.281,15.884,151.927
C06365=1099.751,151.567,-64.434,177.284,15.883,151.927
C06366=1099.757,151.817,-64.455,177.287,15.883,151.926
C06367=1099.763,152.066,-64.475,177.291,15.883,151.925
C06368=1099.768,152.314,-64.497,177.294,15.883,151.924
C06369=1099.774,152.564,-64.518,177.297,15.883,151.924
C06370=1099.780,152.812,-64.539,177.301,15.883,151.923
C06371=1099.786,153.062,-64.560,177.304,15.882,151.922
C06372=1099.791,153.311,-64.581,177.307,15.883,151.922
C06373=1099.796,153.560,-64.602,177.310,15.882,151.921
C06374=1099.803,153.809,-64.623,177.313,15.882,151.920
C06375=1099.808,154.058,-64.644,177.317,15.882,151.920
C06376=1099.813,154.307,-64.665,177.320,15.882,151.919
C06377=1099.819,154.556,-64.686,177.323,15.882,151.918
C06378=1099.825,154.805,-64.707,177.327,15.882,151.917
C06379=1099.831,155.054,-64.729,177.330,15.881,151.916
C06380=1099.836,155.303,-64.749,177.333,15.881,151.916
C06381=1099.841,155.552,-64.771,177.337,15.881,151.915
C06382=1099.847,155.801,-64.793,177.340,15.880,151.914
C06383=1099.852,156.050,-64.813,177.343,15.880,151.914
C06384=1099.859,156.300,-64.835,177.347,15.880,151.913
C06385=1099.864,156.549,-64.856,177.350,15.880,151.912
C06386=1099.869,156.797,-64.877,177.353,15.880,151.911
C06387=1099.876,157.046,-64.899,177.357,15.880,151.911
C06388=1099.881,157.295,-64.920,177.359,15.879,151.910
C06389=1099.887,157.545,-64.941,177.363,15.879,151.909
C06390=1099.892,157.794,-64.963,177.367,15.879,151.908
C06391=1099.897,158.042,-64.984,177.369,15.878,151.908
C06392=1099.903,158.292,-65.005,177.373,15.878,151.907
C06393=1099.909,158.540,-65.026,177.376,15.879,151.906
C06394=1099.915,158.790,-65.048,177.379,15.878,151.906
C06395=1099.921,159.038,-65.069,177.383,15.877,151.905
C06396=1099.926,159.288,-65.090,177.387,15.878,151.904
C06397=1099.931,159.537,-65.112,177.390,15.878,151.903
C06398=1099.938,159.810,-65.135,177.393,15.877,151.902
C06399=1099.944,160.084,-65.158,177.397,15.877,151.902
C06400=1099.951,160.358,-65.182,177.401,15.876,151.901
C06401=1099.957,160.631,-65.207,177.404,15.876,151.900
C06402=1099.962,160.880,-65.227,177.408,15.876,151.899
C06403=1099.968,161.129,-65.249,177.412,15.876,151.898
C06404=1099.974,161.378,-65.270,177.414,15.875,151.898
C06405=1099.979,161.628,-65.292,177.418,15.875,151.897
C06406=1099.985,161.876,-65.313,177.422,15.875,151.896
C06407=1099.991,162.125,-65.335,177.424,15.875,151.895
C06408=1099.996,162.374,-65.357,177.428,15.875,151.895
C06409=1100.001,162.623,-65.378,177.432,15.874,151.894
C06410=1100.006,162.873,-65.400,177.435,15.874,151.893
C06411=1100.012,163.121,-65.421,177.438,15.874,151.892
C06412=1100.017,163.371,-65.443,177.442,15.874,151.892
C06413=1100.023,163.619,-65.465,177.445,15.874,151.891
C06414=1100.029,163.868,-65.486,177.448,15.873,151.890
C06415=1100.034,164.117,-65.508,177.452,15.873,151.889
C06416=1100.040,164.366,-65.530,177.455,15.873,151.889
C06417=1100.045,164.615,-65.552,177.458,15.872,151.888
C06418=1100.051,164.864,-65.573,177.462,15.872,151.887
C06419=1100.056,165.113,-65.595,177.465,15.872,151.886
C06420=1100.062,165.362,-65.617,177.468,15.872,151.886
C06421=1100.067,165.611,-65.639,177.472,15.871,151.885
C06422=1100.073,165.860,-65.660,177.476,15.871,151.884
C06423=1100.078,166.109,-65.682,177.479,15.871,151.883
C06424=1100.084,166.359,-65.704,177.482,15.871,151.883
C06425=1100.089,166.607,-65.726,177.486,15.870,151.882
C06426=1100.095,166.856,-65.748,177.489,15.871,151.881
C06427=1100.100,167.105,-65.770,177.492,15.870,151.880
C06428=1100.106,167.354,-65.791,177.496,15.870,151.880
C06429=1100.112,167.603,-65.814,177.500,15.870,151.879
C06430=1100.117,167.852,-65.835,177.502,15.869,151.878
C06431=1100.123,168.101,-65.857,177.506,15.869,151.877
C06432=1100.128,168.350,-65.878,177.510,15.869,151.876
C06433=1100.134,168.599,-65.901,177.513,15.869,151.876
C06434=1100.140,168.847,-65.923,177.516,15.868,151.875
C06435=1100.145,169.097,-65.945,177.520,15.868,151.874
C06436=1100.151,169.346,-65.966,177.523,15.868,151.873
C06437=1100.156,169.595,-65.988,177.526,15.867,151.873
C06438=1100.163,169.843,-66.011,177.530,15.867,151.872
C06439=1100.167,170.092,-66.033,177.534,15.867,151.871
C06440=1100.173,170.342,-66.055,177.537,15.866,151.870
C06441=1100.179,170.591,-66.076,177.540,15.866,151.869
C06442=1100.184,170.839,-66.099,177.544,15.866,151.869
C06443=1100.190,171.088,-66.121,177.548,15.866,151.868
C06444=1100.196,171.338,-66.143,177.550,15.865,151.867
C06445=1100.202,171.586,-66.165,177.554,15.865,151.866
C06446=1100.207,171.835,-66.187,177.558,15.865,151.865
C06447=1100.212,172.085,-66.209,177.561,15.864,151.865
C06448=1100.218,172.333,-66.231,177.565,15.864,151.864
C06449=1100.224,172.582,-66.254,177.568,15.863,151.863
C06450=1100.230,172.831,-66.275,177.572,15.863,151.862
C06451=1100.235,173.080,-66.298,177.575,15.863,151.861
C06452=1100.240,173.329,-66.320,177.579,15.862,151.861
C06453=1100.247,173.578,-66.342,177.582,15.862,151.860
C06454=1100.252,173.827,-66.365,177.585,15.861,151.859
C06455=1100.257,174.076,-66.386,177.589,15.861,151.858
C06456=1100.264,174.325,-66.409,177.593,15.861,151.857
C06457=1100.269,174.574,-66.431,177.597,15.861,151.856
C06458=1100.274,174.822,-66.454,177.599,15.860,151.856
C06459=1100.280,175.072,-66.475,177.603,15.860,151.855
C06460=1100.286,175.321,-66.497,177.607,15.860,151.854
C06461=1100.291,175.570,-66.520,177.610,15.859,151.853
C06462=1100.298,175.843,-66.545,177.614,15.858,151.852
C06463=1100.304,176.116,-66.569,177.618,15.858,151.851
C06464=1100.310,176.389,-66.593,177.621,15.858,151.851
C06465=1100.316,176.662,-66.618,177.625,15.857,151.850
C06466=1100.322,176.911,-66.640,177.629,15.857,151.849
C06467=1100.328,177.161,-66.663,177.633,15.857,151.848
C06468=1100.334,177.409,-66.686,177.636,15.856,151.847
C06469=1100.340,177.659,-66.707,177.640,15.855,151.846
C06470=1100.345,177.907,-66.730,177.643,15.856,151.846
C06471=1100.350,178.156,-66.752,177.647,15.855,151.845
C06472=1100.356,178.405,-66.775,177.650,15.854,151.844
C06473=1100.362,178.654,-66.797,177.654,15.854,151.843
C06474=1100.368,178.903,-66.820,177.658,15.854,151.842
C06475=1100.374,179.152,-66.843,177.661,15.853,151.841
C06476=1100.379,179.400,-66.865,177.664,15.852,151.840
C06477=1100.385,179.650,-66.887,177.668,15.853,151.840
C06478=1100.391,179.899,-66.910,177.672,15.852,151.839
C06479=1100.396,180.147,-66.933,177.675,15.851,151.838
C06480=1100.402,180.397,-66.955,177.679,15.851,151.837
C06481=1100.408,180.646,-66.977,177.682,15.851,151.836
C06482=1100.414,180.894,-67.000,177.686,15.850,151.835
C06483=1100.419,181.143,-67.023,177.689,15.849,151.835
C06484=1100.425,181.392,-67.045,177.693,15.849,151.834
C06485=1100.430,181.641,-67.068,177.697,15.849,151.833
C06486=1100.437,181.890,-67.090,177.701,15.849,151.832
C06487=1100.442,182.139,-67.113,177.704,15.848,151.831
C06488=1100.448,182.387,-67.136,177.708,15.847,151.830
C06489=1100.454,182.637,-67.158,177.711,15.847,151.829
C06490=1100.459,182.886,-67.181,177.714,15.846,151.829
C06491=1100.466,183.134,-67.204,177.718,15.846,151.828
C06492=1100.472,183.383,-67.227,177.722,15.846,151.827
C06493=1100.477,183.632,-67.250,177.726,15.845,151.826
C06494=1100.483,183.881,-67.273,177.729,15.844,151.825
C06495=1100.488,184.131,-67.295,177.733,15.844,151.824
C06496=1100.494,184.380,-67.318,177.737,15.844,151.823
C06497=1100.500,184.628,-67.341,177.740,15.843,151.823
C06498=1100.506,184.877,-67.363,177.743,15.842,151.822
C06499=1100.512,185.126,-67.386,177.747,15.842,151.821
C06500=1100.517,185.374,-67.409,177.751,15.842,151.820
C06501=1100.523,185.623,-67.432,177.754,15.841,151.819
C06502=1100.528,185.872,-67.455,177.758,15.841,151.818
C06503=1100.534,186.121,-67.478,177.761,15.841,151.818
C06504=1100.539,186.370,-67.501,177.765,15.840,151.817
C06505=1100.545,186.619,-67.524,177.769,15.840,151.816
C06506=1100.551,186.868,-67.547,177.772,15.839,151.815
C06507=1100.557,187.117,-67.570,177.776,15.839,151.814
C06508=1100.562,187.365,-67.592,177.780,15.839,151.813
C06509=1100.567,187.614,-67.616,177.783,15.838,151.812
C06510=1100.572,187.863,-67.639,177.787,15.837,151.812
C06511=1100.578,188.112,-67.662,177.790,15.837,151.811
C06512=1100.584,188.361,-67.685,177.794,15.837,151.810
C06513=1100.590,188.610,-67.708,177.798,15.837,151.809
C06514=1100.595,188.859,-67.731,177.801,15.836,151.808
C06515=1100.600,189.108,-67.754,177.805,15.835,151.807
C06516=1100.606,189.357,-67.777,177.809,15.835,151.806
C06517=1100.612,189.606,-67.800,177.812,15.835,151.806
C06518=1100.618,189.854,-67.823,177.816,15.834,151.805
C06519=1100.623,190.104,-67.847,177.819,15.834,151.804
C06520=1100.629,190.352,-67.870,177.823,15.833,151.803
C06521=1100.634,190.601,-67.893,177.827,15.833,151.802
C06522=1100.640,190.850,-67.916,177.830,15.832,151.801
C06523=1100.645,191.099,-67.940,177.834,15.832,151.800
C06524=1100.651,191.348,-67.963,177.838,15.831,151.800
C06525=1100.657,191.596,-67.986,177.841,15.831,151.799
C06526=1100.662,191.869,-68.011,177.845,15.831,151.798
C06527=1100.668,192.142,-68.037,177.849,15.830,151.797
C06528=1100.675,192.415,-68.062,177.853,15.829,151.796
C06529=1100.681,192.688,-68.088,177.857,15.829,151.795
C06530=1100.687,192.936,-68.111,177.861,15.828,151.794
C06531=1100.692,193.185,-68.135,177.864,15.827,151.793
C06532=1100.698,193.434,-68.158,177.868,15.827,151.792
C06533=1100.704,193.683,-68.181,177.872,15.827,151.791
C06534=1100.709,193.932,-68.205,177.876,15.826,151.790
C06535=1100.715,194.181,-68.228,177.880,15.826,151.790
C06536=1100.721,194.430,-68.251,177.883,15.825,151.789
C06537=1100.726,194.678,-68.275,177.887,15.825,151.788
C06538=1100.732,194.927,-68.298,177.891,15.824,151.787
C06539=1100.737,195.176,-68.321,177.894,15.824,151.786
C06540=1100.743,195.425,-68.345,177.898,15.823,151.785
C06541=1100.749,195.674,-68.369,177.901,15.823,151.784
C06542=1100.755,195.922,-68.392,177.905,15.822,151.783
C06543=1100.760,196.172,-68.416,177.909,15.822,151.783
C06544=1100.766,196.421,-68.439,177.912,15.821,151.782
C06545=1100.772,196.669,-68.462,177.916,15.821,151.781
C06546=1100.777,196.918,-68.486,177.920,15.820,151.780
C06547=1100.783,197.166,-68.510,177.924,15.820,151.779
C06548=1100.788,197.415,-68.533,177.928,15.820,151.778
C06549=1100.794,197.665,-68.557,177.931,15.818,151.777
C06550=1100.800,197.913,-68.580,177.935,15.818,151.776
C06551=1100.805,198.162,-68.604,177.939,15.817,151.775
C06552=1100.811,198.411,-68.627,177.943,15.817,151.774
C06553=1100.817,198.659,-68.651,177.946,15.816,151.774
C06554=1100.823,198.909,-68.675,177.950,15.816,151.773
C06555=1100.829,199.157,-68.699,177.953,15.816,151.772
C06556=1100.834,199.406,-68.723,177.958,15.815,151.771
C06557=1100.840,199.655,-68.746,177.961,15.814,151.770
C06558=1100.846,199.903,-68.770,177.964,15.813,151.769
C06559=1100.851,200.153,-68.793,177.968,15.813,151.768
C06560=1100.858,200.401,-68.817,177.972,15.813,151.767
C06561=1100.863,200.650,-68.841,177.976,15.812,151.766
C06562=1100.869,200.899,-68.864,177.980,15.812,151.765
C06563=1100.874,201.147,-68.889,177.983,15.811,151.765
C06564=1100.880,201.396,-68.913,177.987,15.810,151.764
C06565=1100.885,201.646,-68.936,177.991,15.810,151.763
C06566=1100.891,201.894,-68.960,177.995,15.809,151.762
C06567=1100.898,202.142,-68.983,177.998,15.808,151.761
C06568=1100.903,202.392,-69.007,178.002,15.808,151.760
C06569=1100.909,202.640,-69.031,178.006,15.807,151.759
C06570=1100.914,202.889,-69.055,178.010,15.807,151.758
C06571=1100.920,203.139,-69.079,178.014,15.807,151.757
C06572=1100.926,203.387,-69.103,178.017,15.806,151.756
C06573=1100.931,203.636,-69.127,178.021,15.805,151.755
C06574=1100.937,203.884,-69.151,178.025,15.805,151.754
C06575=1100.943,204.133,-69.175,178.029,15.804,151.753
C06576=1100.948,204.382,-69.199,178.033,15.804,151.753
C06577=1100.954,204.631,-69.223,178.036,15.803,151.752
C06578=1100.960,204.879,-69.247,178.040,15.803,151.751
C06579=1100.965,205.128,-69.271,178.044,15.802,151.750
C06580=1100.971,205.377,-69.296,178.048,15.801,151.749
C06581=1100.977,205.626,-69.319,178.052,15.801,151.748
C06582=1100.982,205.875,-69.343,178.055,15.800,151.747
C06583=1100.988,206.124,-69.368,178.059,15.799,151.746
C06584=1100.994,206.372,-69.391,178.063,15.799,151.745
C06585=1100.999,206.621,-69.415,178.067,15.799,151.744
C06586=1101.004,206.869,-69.440,178.071,15.798,151.743
C06587=1101.011,207.118,-69.464,178.075,15.798,151.742
C06588=1101.016,207.367,-69.488,178.078,15.797,151.742
C06589=1101.022,207.616,-69.512,178.081,15.796,151.741
C06590=1101.045,208.622,-69.610,178.118,15.806,151.735
C06591=1101.053,208.990,-69.646,178.124,15.806,151.734
C06592=1101.062,209.359,-69.682,178.129,15.806,151.733
C06593=1101.070,209.728,-69.719,178.134,15.807,151.732
C06594=1101.078,210.096,-69.755,178.139,15.807,151.731
C06595=1101.085,210.345,-69.779,178.144,15.808,151.730
C06596=1101.090,210.593,-69.804,178.147,15.808,151.730
C06597=1101.095,210.842,-69.828,178.151,15.809,151.729
C06598=1101.101,211.091,-69.852,178.154,15.809,151.728
C06599=1101.106,211.340,-69.877,178.158,15.809,151.728
C06600=1101.113,211.588,-69.902,178.161,15.809,151.727
C06601=1101.118,211.837,-69.926,178.164,15.810,151.726
C06602=1101.123,212.085,-69.951,178.168,15.810,151.726
C06603=1101.129,212.335,-69.975,178.171,15.810,151.725
C06604=1101.135,212.583,-70.000,178.176,15.811,151.724
C06605=1101.141,212.832,-70.025,178.179,15.811,151.723
C06606=1101.146,213.081,-70.049,178.183,15.811,151.723
C06607=1101.152,213.329,-70.074,178.186,15.811,151.722
C06608=1101.157,213.578,-70.099,178.190,15.812,151.721
C06609=1101.163,213.827,-70.123,178.193,15.812,151.721
C06610=1101.169,214.075,-70.148,178.196,15.812,151.720
C06611=1101.173,214.324,-70.173,178.200,15.812,151.719
C06612=1101.179,214.573,-70.198,178.204,15.813,151.719
C06613=1101.185,214.821,-70.223,178.208,15.813,151.718
C06614=1101.191,215.071,-70.247,178.211,15.814,151.717
C06615=1101.196,215.319,-70.272,178.215,15.814,151.717
C06616=1101.202,215.568,-70.297,178.218,15.814,151.716
C06617=1101.208,215.816,-70.321,178.222,15.814,151.715
C06618=1101.213,216.065,-70.347,178.225,15.815,151.715
C06619=1101.218,216.314,-70.371,178.229,15.816,151.714
C06620=1101.225,216.563,-70.397,178.233,15.816,151.713
C06621=1101.230,216.811,-70.421,178.236,15.816,151.713
C06622=1101.236,217.060,-70.446,178.240,15.816,151.712
C06623=1101.241,217.308,-70.470,178.243,15.817,151.711
C06624=1101.247,217.558,-70.496,178.247,15.817,151.711
C06625=1101.252,217.806,-70.521,178.250,15.817,151.710
C06626=1101.258,218.055,-70.546,178.254,15.818,151.709
C06627=1101.264,218.304,-70.571,178.258,15.818,151.709
C06628=1101.270,218.552,-70.596,178.261,15.818,151.708
C06629=1101.275,218.802,-70.621,178.265,15.819,151.707
C06630=1101.281,219.050,-70.646,178.268,15.819,151.707
C06631=1101.287,219.299,-70.670,178.272,15.819,151.706
C06632=1101.292,219.547,-70.695,178.275,15.819,151.705
C06633=1101.298,219.796,-70.721,178.279,15.820,151.705
C06634=1101.304,220.045,-70.746,178.283,15.820,151.704
C06635=1101.309,220.293,-70.771,178.286,15.821,151.703
C06636=1101.315,220.542,-70.796,178.290,15.821,151.703
C06637=1101.320,220.791,-70.821,178.293,15.821,151.702
C06638=1101.326,221.039,-70.846,178.297,15.821,151.701
C06639=1101.332,221.288,-70.872,178.301,15.822,151.700
C06640=1101.338,221.537,-70.896,178.304,15.823,151.700
C06641=1101.343,221.785,-70.922,178.308,15.823,151.699
C06642=1101.349,222.034,-70.947,178.311,15.823,151.698
C06643=1101.358,222.407,-70.985,178.317,15.824,151.697
C06644=1101.366,222.779,-71.023,178.322,15.825,151.696
C06645=1101.374,223.151,-71.061,178.327,15.825,151.695
C06646=1101.382,223.523,-71.099,178.333,15.826,151.695
C06647=1101.388,223.773,-71.123,178.336,15.826,151.694
C06648=1101.394,224.021,-71.149,178.341,15.826,151.693
C06649=1101.399,224.269,-71.174,178.344,15.827,151.693
C06650=1101.405,224.518,-71.200,178.347,15.827,151.692
C06651=1101.411,224.767,-71.225,178.351,15.827,151.691
C06652=1101.416,225.015,-71.250,178.354,15.828,151.691
C06653=1101.422,225.264,-71.276,178.358,15.829,151.690
C06654=1101.428,225.513,-71.301,178.362,15.829,151.689
C06655=1101.433,225.762,-71.327,178.366,15.829,151.688
C06656=1101.439,226.010,-71.352,178.369,15.830,151.688
C06657=1101.444,226.259,-71.378,178.372,15.830,151.687
C06658=1101.450,226.508,-71.403,178.377,15.831,151.686
C06659=1101.455,226.756,-71.429,178.380,15.831,151.686
C06660=1101.462,227.005,-71.454,178.383,15.831,151.685
C06661=1101.467,227.254,-71.480,178.387,15.832,151.685
C06662=1101.473,227.502,-71.505,178.390,15.832,151.684
C06663=1101.478,227.751,-71.531,178.394,15.833,151.683
C06664=1101.484,228.000,-71.556,178.398,15.833,151.683
C06665=1101.490,228.249,-71.582,178.402,15.833,151.682
C06666=1101.495,228.496,-71.607,178.405,15.834,151.681
C06667=1101.501,228.745,-71.633,178.408,15.834,151.681
C06668=1101.506,228.994,-71.659,178.413,15.835,151.680
C06669=1101.512,229.243,-71.684,178.416,15.835,151.679
C06670=1101.518,229.491,-71.711,178.419,15.836,151.679
C06671=1101.524,229.739,-71.736,178.423,15.836,151.678
C06672=1101.529,229.988,-71.762,178.426,15.836,151.677
C06673=1101.536,230.237,-71.787,178.430,15.837,151.677
C06674=1101.541,230.486,-71.813,178.434,15.837,151.676
C06675=1101.546,230.735,-71.839,178.438,15.837,151.675
C06676=1101.552,230.983,-71.864,178.441,15.838,151.675
C06677=1101.558,231.231,-71.891,178.445,15.839,151.674
C06678=1101.563,231.480,-71.917,178.449,15.839,151.673
C06679=1101.569,231.729,-71.943,178.452,15.840,151.673
C06680=1101.575,231.978,-71.968,178.455,15.840,151.672
C06681=1101.580,232.226,-71.994,178.460,15.841,151.671
C06682=1101.586,232.475,-72.020,178.463,15.841,151.671
C06683=1101.591,232.724,-72.046,178.466,15.841,151.670
C06684=1101.597,232.972,-72.071,178.470,15.842,151.669
C06685=1101.603,233.221,-72.097,178.474,15.843,151.669
C06686=1101.608,233.469,-72.124,178.477,15.843,151.668
C06687=1101.613,233.718,-72.150,178.481,15.843,151.667
C06688=1101.620,233.967,-72.175,178.484,15.844,151.667
C06689=1101.625,234.215,-72.202,178.488,15.844,151.666
C06690=1101.631,234.464,-72.228,178.492,15.845,151.666
C06691=1101.636,234.713,-72.253,178.495,15.845,151.665
C06692=1101.642,234.961,-72.280,178.499,15.845,151.664
C06693=1101.647,235.210,-72.306,178.503,15.847,151.664
C06694=1101.653,235.458,-72.332,178.506,15.847,151.663
C06695=1101.661,235.822,-72.370,178.512,15.848,151.662
C06696=1101.669,236.186,-72.409,178.516,15.848,151.661
C06697=1101.678,236.550,-72.446,178.522,15.849,151.660
C06698=1101.686,236.914,-72.485,178.527,15.850,151.659
C06699=1101.691,237.163,-72.511,178.531,15.850,151.659
C06700=1101.697,237.411,-72.538,178.534,15.851,151.658
C06701=1101.703,237.660,-72.563,178.538,15.851,151.657
C06702=1101.709,237.908,-72.590,178.542,15.852,151.657
C06703=1101.715,238.157,-72.616,178.545,15.852,151.656
C06704=1101.720,238.405,-72.642,178.550,15.853,151.655
C06705=1101.726,238.654,-72.668,178.553,15.854,151.655
C06706=1101.732,238.903,-72.695,178.556,15.854,151.654
C06707=1101.737,239.151,-72.721,178.559,15.854,151.654
C06708=1101.743,239.400,-72.747,178.564,15.855,151.653
C06709=1101.749,239.648,-72.774,178.567,15.855,151.652
C06710=1101.753,239.897,-72.800,178.571,15.856,151.652
C06711=1101.759,240.145,-72.826,178.575,15.857,151.651
C06712=1101.765,240.393,-72.853,178.578,15.857,151.650
C06713=1101.770,240.642,-72.879,178.582,15.858,151.650
C06714=1101.776,240.891,-72.905,178.585,15.858,151.649
C06715=1101.782,241.139,-72.932,178.589,15.859,151.648
C06716=1101.787,241.388,-72.958,178.593,15.859,151.648
C06717=1101.793,241.636,-72.985,178.596,15.860,151.647
C06718=1101.799,241.885,-73.011,178.600,15.861,151.646
C06719=1101.805,242.133,-73.038,178.604,15.861,151.646
C06720=1101.811,242.383,-73.064,178.607,15.862,151.645
C06721=1101.817,242.631,-73.091,178.610,15.862,151.644
C06722=1101.822,242.880,-73.118,178.614,15.863,151.644
C06723=1101.828,243.128,-73.144,178.618,15.863,151.643
C06724=1101.834,243.376,-73.171,178.622,15.863,151.643
C06725=1101.839,243.626,-73.197,178.625,15.865,151.642
C06726=1101.844,243.874,-73.224,178.629,15.865,151.641
C06727=1101.850,244.122,-73.251,178.632,15.865,151.641
C06728=1101.856,244.371,-73.277,178.637,15.866,151.640
C06729=1101.862,244.619,-73.304,178.640,15.867,151.640
C06730=1101.867,244.868,-73.331,178.643,15.867,151.639
C06731=1101.872,245.117,-73.357,178.647,15.868,151.638
C06732=1101.878,245.365,-73.384,178.651,15.868,151.638
C06733=1101.884,245.613,-73.410,178.654,15.869,151.637
C06734=1101.890,245.862,-73.437,178.658,15.870,151.636
C06735=1101.895,246.110,-73.464,178.662,15.871,151.636
C06736=1101.900,246.359,-73.491,178.665,15.871,151.635
C06737=1101.906,246.607,-73.518,178.669,15.872,151.635
C06738=1101.912,246.855,-73.544,178.672,15.873,151.634
C06739=1101.917,247.104,-73.572,178.676,15.873,151.633
C06740=1101.923,247.353,-73.599,178.680,15.874,151.633
C06741=1101.929,247.602,-73.625,178.683,15.874,151.632
C06742=1101.934,247.850,-73.652,178.687,15.875,151.632
C06743=1101.940,248.099,-73.679,178.691,15.876,151.631
C06744=1101.946,248.347,-73.706,178.694,15.876,151.630
C06745=1101.951,248.596,-73.733,178.697,15.877,151.630
C06746=1101.957,248.844,-73.760,178.702,15.878,151.629
C06747=1101.964,249.201,-73.798,178.706,15.878,151.628
C06748=1101.972,249.558,-73.838,178.712,15.879,151.627
C06749=1101.981,249.915,-73.877,178.717,15.880,151.626
C06750=1101.989,250.272,-73.915,178.722,15.882,151.626
C06751=1101.994,250.521,-73.942,178.726,15.882,151.625
C06752=1101.999,250.769,-73.969,178.730,15.883,151.624
C06753=1102.005,251.018,-73.996,178.733,15.883,151.624
C06754=1102.011,251.266,-74.024,178.736,15.884,151.623
C06755=1102.017,251.515,-74.051,178.740,15.885,151.623
C06756=1102.022,251.764,-74.078,178.744,15.886,151.622
C06757=1102.028,252.012,-74.105,178.747,15.886,151.621
C06758=1102.033,252.260,-74.133,178.751,15.887,151.621
C06759=1102.039,252.508,-74.159,178.754,15.888,151.620
C06760=1102.044,252.757,-74.187,178.758,15.889,151.620
C06761=1102.051,253.005,-74.214,178.762,15.889,151.619
C06762=1102.056,253.254,-74.242,178.765,15.890,151.618
C06763=1102.061,253.503,-74.268,178.769,15.891,151.618
C06764=1102.066,253.751,-74.296,178.773,15.891,151.617
C06765=1102.072,253.999,-74.323,178.776,15.892,151.617
C06766=1102.078,254.248,-74.351,178.780,15.893,151.616
C06767=1102.084,254.496,-74.378,178.783,15.893,151.615
C06768=1102.089,254.745,-74.405,178.787,15.895,151.615
C06769=1102.095,254.993,-74.432,178.791,15.895,151.614
C06770=1102.101,255.242,-74.460,178.794,15.895,151.614
C06771=1102.106,255.490,-74.487,178.798,15.897,151.613
C06772=1102.112,255.738,-74.515,178.802,15.897,151.612
C06773=1102.117,255.987,-74.542,178.806,15.898,151.612
C06774=1102.124,256.235,-74.570,178.809,15.898,151.611
C06775=1102.129,256.484,-74.597,178.812,15.899,151.611
C06776=1102.135,256.732,-74.624,178.816,15.900,151.610
C06777=1102.141,256.981,-74.652,178.820,15.901,151.609
C06778=1102.146,257.229,-74.680,178.823,15.901,151.609
C06779=1102.152,257.478,-74.706,178.827,15.902,151.608
C06780=1102.158,257.726,-74.735,178.831,15.903,151.608
C06781=1102.163,257.975,-74.762,178.835,15.904,151.607
C06782=1102.169,258.223,-74.789,178.838,15.904,151.606
C06783=1102.175,258.471,-74.818,178.841,15.905,151.606
C06784=1102.180,258.720,-74.844,178.845,15.906,151.605
C06785=1102.186,258.968,-74.872,178.849,15.906,151.605
C06786=1102.191,259.217,-74.900,178.853,15.908,151.604
C06787=1102.197,259.465,-74.927,178.856,15.908,151.604
C06788=1102.203,259.713,-74.955,178.860,15.908,151.603
C06789=1102.208,259.962,-74.983,178.864,15.910,151.602
C06790=1102.215,260.210,-75.010,178.867,15.910,151.602
C06791=1102.220,260.458,-75.038,178.871,15.911,151.601
C06792=1102.226,260.707,-75.067,178.874,15.912,151.601
C06793=1102.232,260.955,-75.093,178.878,15.913,151.600
C06794=1102.238,261.204,-75.122,178.882,15.913,151.599
C06795=1102.243,261.452,-75.149,178.885,15.914,151.599
C06796=1102.249,261.701,-75.178,178.889,15.915,151.598
C06797=1102.255,261.949,-75.204,178.893,15.915,151.598
C06798=1102.260,262.197,-75.232,178.897,15.917,151.597
C06799=1102.269,262.551,-75.272,178.902,15.918,151.596
C06800=1102.277,262.907,-75.312,178.906,15.918,151.595
C06801=1102.285,263.260,-75.351,178.912,15.919,151.595
C06802=1102.293,263.614,-75.392,178.917,15.921,151.594
C06803=1102.299,263.862,-75.419,178.921,15.922,151.593
C06804=1102.305,264.111,-75.448,178.924,15.922,151.593
C06805=1102.310,264.360,-75.475,178.928,15.923,151.592
C06806=1102.316,264.608,-75.503,178.932,15.924,151.591
C06807=1102.321,264.856,-75.531,178.935,15.925,151.591
C06808=1102.327,265.105,-75.559,178.939,15.926,151.590
C06809=1102.333,265.353,-75.587,178.942,15.926,151.590
C06810=1102.339,265.602,-75.616,178.946,15.928,151.589
C06811=1102.344,265.850,-75.644,178.950,15.928,151.589
C06812=1102.350,266.099,-75.672,178.954,15.929,151.588
C06813=1102.355,266.347,-75.700,178.957,15.930,151.588
C06814=1102.361,266.595,-75.727,178.961,15.931,151.587
C06815=1102.367,266.843,-75.756,178.964,15.932,151.586
C06816=1102.373,267.091,-75.784,178.967,15.933,151.586
C06817=1102.378,267.340,-75.812,178.972,15.933,151.585
C06818=1102.384,267.588,-75.840,178.975,15.934,151.585
C06819=1102.390,267.836,-75.869,178.979,15.935,151.584
C06820=1102.395,268.084,-75.897,178.982,15.936,151.584
C06821=1102.401,268.333,-75.926,178.986,15.937,151.583
C06822=1102.406,268.582,-75.954,178.989,15.938,151.583
C06823=1102.412,268.830,-75.982,178.993,15.939,151.582
C06824=1102.417,269.078,-76.010,178.997,15.939,151.581
C06825=1102.423,269.327,-76.038,179.001,15.941,151.581
C06826=1102.429,269.574,-76.067,179.004,15.941,151.580
C06827=1102.435,269.823,-76.095,179.008,15.943,151.580
C06828=1102.441,270.072,-76.124,179.011,15.943,151.579
C06829=1102.446,270.320,-76.152,179.015,15.945,151.579
C06830=1102.452,270.568,-76.181,179.018,15.945,151.578
C06831=1102.458,270.816,-76.209,179.022,15.947,151.578
C06832=1102.464,271.065,-76.237,179.025,15.947,151.577
C06833=1102.468,271.313,-76.266,179.030,15.948,151.577
C06834=1102.474,271.561,-76.295,179.033,15.949,151.576
C06835=1102.480,271.810,-76.323,179.036,15.949,151.575
C06836=1102.486,272.058,-76.351,179.040,15.951,151.575
C06837=1102.492,272.306,-76.380,179.043,15.951,151.574
C06838=1102.497,272.554,-76.408,179.047,15.953,151.574
C06839=1102.503,272.804,-76.437,179.051,15.953,151.573
C06840=1102.508,273.051,-76.466,179.055,15.955,151.573
C06841=1102.514,273.300,-76.494,179.058,15.955,151.572
C06842=1102.520,273.548,-76.522,179.062,15.957,151.572
C06843=1102.526,273.796,-76.551,179.065,15.957,151.571
C06844=1102.531,274.045,-76.580,179.069,15.959,151.571
C06845=1102.537,274.292,-76.608,179.073,15.960,151.570
C06846=1102.542,274.541,-76.637,179.076,15.961,151.570
C06847=1102.549,274.789,-76.666,179.080,15.962,151.569
C06848=1102.553,275.038,-76.694,179.083,15.963,151.569
C06849=1102.560,275.286,-76.723,179.087,15.964,151.568
C06850=1102.565,275.534,-76.751,179.090,15.964,151.568
C06851=1102.573,275.892,-76.793,179.096,15.966,151.567
C06852=1102.581,276.249,-76.834,179.101,15.967,151.566
C06853=1102.590,276.605,-76.876,179.106,15.969,151.565
C06854=1102.597,276.963,-76.917,179.111,15.970,151.565
C06855=1102.603,277.211,-76.946,179.115,15.971,151.564
C06856=1102.609,277.459,-76.976,179.118,15.972,151.564
C06857=1102.614,277.707,-77.004,179.122,15.973,151.563
C06858=1102.620,277.955,-77.033,179.126,15.975,151.563
C06859=1102.626,278.204,-77.062,179.129,15.975,151.562
C06860=1102.631,278.452,-77.090,179.133,15.977,151.562
C06861=1102.637,278.700,-77.120,179.136,15.977,151.561
C06862=1102.643,278.948,-77.149,179.140,15.979,151.561
C06863=1102.648,279.196,-77.177,179.143,15.980,151.560
C06864=1102.654,279.445,-77.207,179.147,15.981,151.560
C06865=1102.660,279.693,-77.236,179.151,15.982,151.559
C06866=1102.666,279.941,-77.265,179.154,15.983,151.559
C06867=1102.671,280.189,-77.293,179.158,15.984,151.558
C06868=1102.677,280.438,-77.323,179.162,15.985,151.558
C06869=1102.683,280.686,-77.352,179.166,15.986,151.557
C06870=1102.688,280.934,-77.381,179.169,15.987,151.556
C06871=1102.694,281.182,-77.410,179.172,15.989,151.556
C06872=1102.699,281.431,-77.439,179.176,15.989,151.556
C06873=1102.705,281.679,-77.468,179.180,15.991,151.555
C06874=1102.710,281.927,-77.498,179.183,15.991,151.555
C06875=1102.717,282.175,-77.527,179.187,15.993,151.554
C06876=1102.722,282.423,-77.556,179.190,15.994,151.554
C06877=1102.728,282.672,-77.586,179.194,15.995,151.553
C06878=1102.733,282.919,-77.615,179.198,15.996,151.553
C06879=1102.739,283.168,-77.644,179.201,15.997,151.552
C06880=1102.745,283.416,-77.673,179.205,15.999,151.552
C06881=1102.750,283.665,-77.702,179.208,16.000,151.551
C06882=1102.755,283.913,-77.731,179.212,16.001,151.551
C06883=1102.761,284.161,-77.760,179.216,16.002,151.550
C06884=1102.767,284.409,-77.790,179.219,16.003,151.550
C06885=1102.772,284.658,-77.820,179.223,16.005,151.549
C06886=1102.779,284.906,-77.849,179.226,16.005,151.549
C06887=1102.784,285.154,-77.878,179.229,16.007,151.548
C06888=1102.789,285.401,-77.908,179.233,16.008,151.548
C06889=1102.796,285.650,-77.937,179.237,16.009,151.547
C06890=1102.801,285.898,-77.967,179.241,16.010,151.547
C06891=1102.807,286.146,-77.997,179.243,16.011,151.547
C06892=1102.813,286.395,-78.026,179.247,16.013,151.546
C06893=1102.818,286.642,-78.055,179.251,16.013,151.546
C06894=1102.823,286.891,-78.085,179.254,16.015,151.545
C06895=1102.829,287.139,-78.114,179.258,16.016,151.545
C06896=1102.835,287.387,-78.143,179.261,16.017,151.544
C06897=1102.841,287.635,-78.174,179.265,16.018,151.544
C06898=1102.846,287.884,-78.203,179.268,16.020,151.543
C06899=1102.852,288.132,-78.233,179.272,16.021,151.543
C06900=1102.858,288.379,-78.262,179.276,16.022,151.542
C06901=1102.863,288.628,-78.291,179.279,16.023,151.542
C06902=1102.869,288.876,-78.322,179.283,16.025,151.541
C06903=1102.878,289.242,-78.365,179.288,16.026,151.541
C06904=1102.886,289.609,-78.409,179.294,16.028,151.540
C06905=1102.895,289.975,-78.453,179.299,16.030,151.539
C06906=1102.903,290.342,-78.497,179.304,16.032,151.539
C06907=1102.908,290.590,-78.527,179.308,16.033,151.538
C06908=1102.914,290.839,-78.556,179.312,16.035,151.538
C06909=1102.920,291.086,-78.586,179.315,16.036,151.537
C06910=1102.925,291.335,-78.616,179.319,16.037,151.537
C06911=1102.931,291.583,-78.646,179.322,16.039,151.537
C06912=1102.937,291.831,-78.676,179.325,16.039,151.536
C06913=1102.943,292.079,-78.705,179.329,16.041,151.536
C06914=1102.949,292.327,-78.736,179.332,16.042,151.535
C06915=1102.953,292.575,-78.765,179.336,16.044,151.535
C06916=1102.959,292.823,-78.795,179.340,16.045,151.534
C06917=1102.965,293.071,-78.825,179.343,16.046,151.534
C06918=1102.971,293.319,-78.855,179.347,16.047,151.533
C06919=1102.976,293.567,-78.885,179.350,16.049,151.533
C06920=1102.982,293.815,-78.915,179.354,16.050,151.533
C06921=1102.987,294.064,-78.945,179.357,16.051,151.532
C06922=1102.993,294.311,-78.975,179.361,16.053,151.532
C06923=1102.999,294.560,-79.005,179.364,16.054,151.531
C06924=1103.005,294.808,-79.035,179.368,16.056,151.531
C06925=1103.010,295.055,-79.065,179.372,16.057,151.531
C06926=1103.016,295.304,-79.095,179.375,16.058,151.530
C06927=1103.022,295.552,-79.125,179.379,16.059,151.530
C06928=1103.027,295.800,-79.155,179.382,16.061,151.529
C06929=1103.033,296.048,-79.185,179.385,16.062,151.529
C06930=1103.039,296.296,-79.216,179.389,16.064,151.528
C06931=1103.044,296.545,-79.246,179.393,16.065,151.528
C06932=1103.050,296.792,-79.276,179.396,16.066,151.528
C06933=1103.055,297.040,-79.307,179.400,16.068,151.527
C06934=1103.061,297.288,-79.337,179.404,16.069,151.527
C06935=1103.067,297.536,-79.367,179.407,16.071,151.526
C06936=1103.073,297.785,-79.397,179.410,16.072,151.526
C06937=1103.079,298.033,-79.428,179.414,16.073,151.526
C06938=1103.085,298.281,-79.458,179.418,16.075,151.525
C06939=1103.089,298.529,-79.488,179.421,16.076,151.525
C06940=1103.095,298.777,-79.519,179.424,16.078,151.524
C06941=1103.101,299.025,-79.549,179.428,16.079,151.524
C06942=1103.106,299.273,-79.580,179.432,16.081,151.524
C06943=1103.112,299.521,-79.610,179.435,16.082,151.523
C06944=1103.118,299.769,-79.640,179.439,16.084,151.523
C06945=1103.123,300.017,-79.670,179.442,16.086,151.523
C06946=1103.128,300.265,-79.701,179.445,16.087,151.522
C06947=1103.134,300.513,-79.732,179.449,16.088,151.522
C06948=1103.140,300.761,-79.762,179.453,16.090,151.521
C06949=1103.145,301.009,-79.793,179.456,16.092,151.521
C06950=1103.151,301.257,-79.823,179.459,16.093,151.521
C06951=1103.157,301.505,-79.854,179.463,16.094,151.520
C06952=1103.162,301.753,-79.885,179.467,16.096,151.520
C06953=1103.168,302.001,-79.915,179.470,16.098,151.520
C06954=1103.173,302.249,-79.946,179.473,16.099,151.519
C06955=1103.182,302.629,-79.992,179.479,16.101,151.519
C06956=1103.191,303.010,-80.040,179.484,16.104,151.518
C06957=1103.199,303.391,-80.086,179.490,16.107,151.518
C06958=1103.208,303.771,-80.133,179.495,16.109,151.517
C06959=1103.213,304.019,-80.164,179.498,16.110,151.517
C06960=1103.219,304.267,-80.195,179.502,16.112,151.516
C06961=1103.224,304.515,-80.226,179.506,16.114,151.516
C06962=1103.230,304.763,-80.256,179.509,16.115,151.516
C06963=1103.236,305.011,-80.288,179.512,16.116,151.515
C06964=1103.242,305.259,-80.318,179.516,16.118,151.515
C06965=1103.247,305.506,-80.349,179.520,16.120,151.515
C06966=1103.252,305.755,-80.380,179.523,16.122,151.514
C06967=1103.258,306.002,-80.410,179.526,16.123,151.514
C06968=1103.264,306.251,-80.442,179.530,16.124,151.513
C06969=1103.270,306.498,-80.472,179.534,16.126,151.513
C06970=1103.275,306.747,-80.503,179.537,16.128,151.513
C06971=1103.281,306.994,-80.534,179.541,16.130,151.512
C06972=1103.286,307.242,-80.565,179.544,16.131,151.512
C06973=1103.293,307.490,-80.596,179.547,16.133,151.512
C06974=1103.298,307.739,-80.627,179.551,16.134,151.511
C06975=1103.304,307.986,-80.657,179.555,16.136,151.511
C06976=1103.309,308.234,-80.689,179.558,16.137,151.511
C06977=1103.315,308.482,-80.720,179.561,16.139,151.510
C06978=1103.321,308.731,-80.751,179.565,16.141,151.510
C06979=1103.327,308.978,-80.782,179.569,16.142,151.510
C06980=1103.332,309.227,-80.813,179.572,16.144,151.509
C06981=1103.338,309.474,-80.845,179.575,16.146,151.509
C06982=1103.344,309.722,-80.875,179.578,16.148,151.509
C06983=1103.349,309.971,-80.906,179.582,16.149,151.509
C06984=1103.355,310.218,-80.937,179.586,16.151,151.508
C06985=1103.360,310.466,-80.968,179.589,16.153,151.508
C06986=1103.366,310.714,-81.000,179.592,16.154,151.507
C06987=1103.372,310.962,-81.031,179.596,16.156,151.507
C06988=1103.378,311.210,-81.062,179.600,16.157,151.507
C06989=1103.384,311.458,-81.093,179.603,16.159,151.506
C06990=1103.389,311.706,-81.125,179.607,16.161,151.506
C06991=1103.395,311.954,-81.156,179.610,16.163,151.506
C06992=1103.401,312.202,-81.187,179.613,16.164,151.506
C06993=1103.406,312.450,-81.218,179.617,16.166,151.505
C06994=1103.412,312.698,-81.250,179.620,16.168,151.505
C06995=1103.418,312.945,-81.281,179.624,16.170,151.505
C06996=1103.423,313.193,-81.312,179.628,16.171,151.504
C06997=1103.430,313.441,-81.343,179.630,16.173,151.504
C06998=1103.435,313.689,-81.374,179.634,16.175,151.504
C06999=1103.441,313.938,-81.406,179.638,16.176,151.503
C07000=1103.447,314.185,-81.438,179.641,16.178,151.503
C07001=1103.453,314.434,-81.469,179.645,16.180,151.503
C07002=1103.458,314.681,-81.500,179.648,16.181,151.503
C07003=1103.464,314.929,-81.533,179.651,16.183,151.502
C07004=1103.471,315.177,-81.564,179.655,16.185,151.502
C07005=1103.476,315.425,-81.595,179.659,16.187,151.502
C07006=1103.482,315.673,-81.627,179.662,16.189,151.501
C07007=1103.489,316.056,-81.675,179.667,16.192,151.501
C07008=1103.499,316.438,-81.724,179.673,16.195,151.501
C07009=1103.507,316.822,-81.773,179.678,16.198,151.500
C07010=1103.515,317.205,-81.822,179.683,16.201,151.500
C07011=1103.521,317.453,-81.854,179.686,16.203,151.499
C07012=1103.527,317.700,-81.886,179.690,16.205,151.499
C07013=1103.532,317.948,-81.917,179.693,16.206,151.499
C07014=1103.538,318.196,-81.949,179.696,16.208,151.499
C07015=1103.543,318.444,-81.980,179.699,16.210,151.499
C07016=1103.549,318.692,-82.012,179.703,16.212,151.498
C07017=1103.554,318.940,-82.044,179.706,16.214,151.498
C07018=1103.560,319.188,-82.076,179.710,16.216,151.498
C07019=1103.566,319.436,-82.108,179.713,16.218,151.498
C07020=1103.572,319.684,-82.140,179.717,16.220,151.497
C07021=1103.577,319.931,-82.171,179.720,16.222,151.497
C07022=1103.583,320.180,-82.203,179.723,16.224,151.497
C07023=1103.589,320.427,-82.235,179.726,16.226,151.497
C07024=1103.595,320.675,-82.267,179.730,16.228,151.496
C07025=1103.600,320.923,-82.299,179.733,16.230,151.496
C07026=1103.605,321.171,-82.331,179.737,16.232,151.496
C07027=1103.611,321.419,-82.363,179.740,16.234,151.496
C07028=1103.617,321.667,-82.395,179.744,16.236,151.496
C07029=1103.622,321.915,-82.427,179.747,16.238,151.495
C07030=1103.628,322.163,-82.459,179.751,16.240,151.495
C07031=1103.633,322.410,-82.490,179.754,16.242,151.495
C07032=1103.639,322.659,-82.522,179.757,16.244,151.495
C07033=1103.646,322.906,-82.555,179.761,16.246,151.495
C07034=1103.650,323.154,-82.587,179.764,16.247,151.494
C07035=1103.656,323.402,-82.619,179.767,16.250,151.494
C07036=1103.662,323.650,-82.651,179.770,16.252,151.494
C07037=1103.668,323.898,-82.683,179.774,16.254,151.494
C07038=1103.674,324.146,-82.715,179.777,16.256,151.494
C07039=1103.679,324.393,-82.748,179.781,16.258,151.493
C07040=1103.685,324.642,-82.780,179.784,16.260,151.493
C07041=1103.690,324.889,-82.812,179.787,16.262,151.493
C07042=1103.696,325.137,-82.844,179.791,16.265,151.493
C07043=1103.702,325.385,-82.877,179.794,16.267,151.493
C07044=1103.707,325.633,-82.909,179.798,16.268,151.492
C07045=1103.713,325.881,-82.941,179.801,16.271,151.492
C07046=1103.719,326.129,-82.974,179.804,16.273,151.492
C07047=1103.725,326.376,-83.005,179.808,16.275,151.492
C07048=1103.730,326.625,-83.038,179.811,16.277,151.492
C07049=1103.736,326.872,-83.071,179.814,16.279,151.491
C07050=1103.741,327.120,-83.102,179.818,16.282,151.491
C07051=1103.747,327.368,-83.134,179.821,16.284,151.491
C07052=1103.753,327.616,-83.168,179.825,16.286,151.491
C07053=1103.759,327.864,-83.200,179.828,16.288,151.491
C07054=1103.765,328.111,-83.232,179.831,16.290,151.490
C07055=1103.771,328.359,-83.264,179.835,16.292,151.490
C07056=1103.776,328.608,-83.297,179.838,16.294,151.490
C07057=1103.782,328.855,-83.329,179.841,16.296,151.490
C07058=1103.788,329.103,-83.361,179.845,16.299,151.490
C07059=1103.796,329.478,-83.411,179.850,16.302,151.490
C07060=1103.805,329.854,-83.461,179.855,16.305,151.489
C07061=1103.814,330.230,-83.510,179.860,16.309,151.489
C07062=1103.822,330.607,-83.559,179.865,16.312,151.489
C07063=1103.828,330.853,-83.592,179.868,16.314,151.489
C07064=1103.834,331.102,-83.624,179.872,16.316,151.488
C07065=1103.840,331.350,-83.657,179.875,16.318,151.488
C07066=1103.846,331.597,-83.690,179.878,16.321,151.488
C07067=1103.851,331.846,-83.723,179.882,16.323,151.488
C07068=1103.858,332.093,-83.755,179.885,16.325,151.488
C07069=1103.863,332.340,-83.788,179.888,16.327,151.488
C07070=1103.869,332.589,-83.820,179.891,16.330,151.488
C07071=1103.874,332.837,-83.854,179.895,16.332,151.487
C07072=1103.880,333.084,-83.886,179.898,16.334,151.487
C07073=1103.886,333.333,-83.919,179.901,16.337,151.487
C07074=1103.891,333.580,-83.951,179.904,16.339,151.487
C07075=1103.897,333.828,-83.985,179.907,16.341,151.487
C07076=1103.902,334.075,-84.018,179.911,16.344,151.487
C07077=1103.908,334.324,-84.050,179.914,16.346,151.487
C07078=1103.914,334.572,-84.083,179.918,16.349,151.487
C07079=1103.920,334.818,-84.116,179.921,16.351,151.487
C07080=1103.925,335.066,-84.149,179.924,16.354,151.487
C07081=1103.931,335.314,-84.182,179.928,16.356,151.486
C07082=1103.937,335.562,-84.214,179.931,16.358,151.486
C07083=1103.942,335.810,-84.248,179.934,16.361,151.486
C07084=1103.948,336.058,-84.281,179.937,16.363,151.486
C07085=1103.954,336.305,-84.314,179.940,16.366,151.486
C07086=1103.959,336.553,-84.347,179.944,16.368,151.486
C07087=1103.965,336.801,-84.380,179.947,16.370,151.486
C07088=1103.971,337.049,-84.413,179.950,16.373,151.486
C07089=1103.976,337.296,-84.446,179.954,16.376,151.486
C07090=1103.982,337.544,-84.480,179.957,16.378,151.486
C07091=1103.988,337.792,-84.512,179.960,16.381,151.486
C07092=1103.994,338.040,-84.546,179.964,16.383,151.485
C07093=1103.999,338.288,-84.579,179.967,16.385,151.485
C07094=1104.005,338.536,-84.612,179.970,16.388,151.485
C07095=1104.011,338.783,-84.645,179.973,16.390,151.485
C07096=1104.016,339.030,-84.678,179.976,16.393,151.485
C07097=1104.022,339.278,-84.711,179.980,16.395,151.485
C07098=1104.027,339.526,-84.745,179.983,16.398,151.485
C07099=1104.033,339.774,-84.778,179.986,16.401,151.485
C07100=1104.038,340.022,-84.811,179.989,16.403,151.485
C07101=1104.045,340.269,-84.845,179.993,16.406,151.485
C07102=1104.051,340.517,-84.878,179.996,16.408,151.485
C07103=1104.056,340.765,-84.912,179.999,16.411,151.485
C07104=1104.062,341.013,-84.945,-179.997,16.414,151.485
C07105=1104.067,341.261,-84.978,-179.994,16.417,151.485
C07106=1104.073,341.509,-85.012,-179.991,16.419,151.485
C07107=1104.079,341.756,-85.046,-179.988,16.421,151.485
C07108=1104.084,342.004,-85.079,-179.985,16.424,151.485
C07109=1104.090,342.252,-85.112,-179.982,16.427,151.485
C07110=1104.095,342.499,-85.145,-179.978,16.430,151.485
C07111=1104.104,342.868,-85.196,-179.973,16.434,151.485
C07112=1104.113,343.239,-85.246,-179.969,16.437,151.485
C07113=1104.121,343.608,-85.296,-179.964,16.441,151.485
C07114=1104.130,343.978,-85.345,-179.959,16.446,151.485
C07115=1104.135,344.226,-85.379,-179.956,16.448,151.485
C07116=1104.141,344.473,-85.413,-179.953,16.451,151.485
C07117=1104.147,344.721,-85.446,-179.949,16.453,151.485
C07118=1104.153,344.968,-85.480,-179.946,16.456,151.485
C07119=1104.158,345.216,-85.514,-179.943,16.459,151.485
C07120=1104.164,345.463,-85.548,-179.940,16.462,151.485
C07121=1104.170,345.711,-85.581,-179.937,16.464,151.485
C07122=1104.175,345.959,-85.614,-179.934,16.467,151.485
C07123=1104.180,346.207,-85.649,-179.930,16.471,151.485
C07124=1104.186,346.455,-85.682,-179.927,16.473,151.485
C07125=1104.192,346.702,-85.716,-179.924,16.476,151.485
C07126=1104.198,346.949,-85.750,-179.921,16.478,151.485
C07127=1104.203,347.197,-85.784,-179.918,16.481,151.485
C07128=1104.210,347.445,-85.818,-179.914,16.485,151.485
C07129=1104.215,347.693,-85.851,-179.911,16.487,151.485
C07130=1104.221,347.940,-85.885,-179.908,16.490,151.485
C07131=1104.226,348.188,-85.919,-179.905,16.493,151.485
C07132=1104.232,348.436,-85.953,-179.902,16.496,151.485
C07133=1104.238,348.683,-85.988,-179.899,16.499,151.485
C07134=1104.243,348.931,-86.021,-179.896,16.501,151.485
C07135=1104.249,349.178,-86.055,-179.892,16.505,151.485
C07136=1104.254,349.426,-86.090,-179.889,16.507,151.485
C07137=1104.260,349.674,-86.123,-179.886,16.510,151.485
C07138=1104.266,349.921,-86.157,-179.883,16.513,151.485
C07139=1104.272,350.169,-86.191,-179.879,16.516,151.485
C07140=1104.277,350.417,-86.226,-179.877,16.519,151.486
C07141=1104.283,350.664,-86.259,-179.874,16.522,151.486
C07142=1104.289,350.912,-86.293,-179.870,16.526,151.486
C07143=1104.294,351.159,-86.327,-179.867,16.528,151.486
C07144=1104.300,351.407,-86.362,-179.864,16.531,151.486
C07145=1104.305,351.655,-86.395,-179.861,16.534,151.486
C07146=1104.312,351.903,-86.430,-179.858,16.537,151.486
C07147=1104.317,352.150,-86.464,-179.855,16.540,151.486
C07148=1104.323,352.397,-86.499,-179.852,16.543,151.486
C07149=1104.328,352.645,-86.533,-179.848,16.547,151.487
C07150=1104.334,352.892,-86.567,-179.845,16.549,151.487
C07151=1104.340,353.140,-86.602,-179.843,16.552,151.487
C07152=1104.346,353.388,-86.636,-179.839,16.555,151.487
C07153=1104.352,353.635,-86.670,-179.836,16.558,151.487
C07154=1104.357,353.882,-86.704,-179.833,16.561,151.487
C07155=1104.363,354.130,-86.739,-179.830,16.565,151.487
C07156=1104.368,354.377,-86.773,-179.827,16.568,151.487
C07157=1104.374,354.625,-86.808,-179.824,16.571,151.487
C07158=1104.379,354.873,-86.842,-179.820,16.574,151.488
C07159=1104.385,355.120,-86.876,-179.818,16.577,151.488
C07160=1104.391,355.367,-86.910,-179.814,16.581,151.488
C07161=1104.397,355.616,-86.945,-179.811,16.584,151.488
C07162=1104.403,355.863,-86.979,-179.809,16.587,151.488
C07163=1104.411,356.235,-87.031,-179.804,16.592,151.488
C07164=1104.419,356.607,-87.082,-179.799,16.596,151.489
C07165=1104.428,356.978,-87.135,-179.795,16.601,151.489
C07166=1104.436,357.351,-87.186,-179.790,16.606,151.489
C07167=1104.442,357.598,-87.221,-179.787,16.609,151.489
C07168=1104.448,357.846,-87.256,-179.784,16.612,151.489
C07169=1104.453,358.093,-87.291,-179.781,16.616,151.490
C07170=1104.459,358.341,-87.326,-179.778,16.619,151.490
C07171=1104.465,358.589,-87.360,-179.775,16.623,151.490
C07172=1104.470,358.836,-87.395,-179.772,16.626,151.490
C07173=1104.476,359.083,-87.429,-179.769,16.629,151.490
C07174=1104.481,359.331,-87.464,-179.766,16.633,151.491
C07175=1104.488,359.579,-87.498,-179.763,16.636,151.491
C07176=1104.493,359.826,-87.534,-179.759,16.639,151.491
C07177=1104.498,360.073,-87.568,-179.757,16.642,151.491
C07178=1104.505,360.321,-87.603,-179.753,16.646,151.491
C07179=1104.510,360.568,-87.638,-179.751,16.649,151.492
C07180=1104.516,360.816,-87.672,-179.748,16.652,151.492
C07181=1104.522,361.063,-87.708,-179.745,16.656,151.492
C07182=1104.527,361.311,-87.743,-179.742,16.659,151.492
C07183=1104.532,361.558,-87.777,-179.738,16.663,151.492
C07184=1104.539,361.806,-87.812,-179.736,16.666,151.493
C07185=1104.544,362.053,-87.847,-179.732,16.670,151.493
C07186=1104.550,362.300,-87.882,-179.730,16.673,151.493
C07187=1104.556,362.548,-87.917,-179.726,16.677,151.493
C07188=1104.562,362.795,-87.952,-179.724,16.680,151.494
C07189=1104.567,363.043,-87.987,-179.720,16.684,151.494
C07190=1104.573,363.291,-88.023,-179.718,16.687,151.494
C07191=1104.579,363.538,-88.057,-179.715,16.691,151.494
C07192=1104.585,363.785,-88.092,-179.712,16.695,151.495
C07193=1104.590,364.032,-88.128,-179.709,16.698,151.495
C07194=1104.595,364.280,-88.162,-179.706,16.702,151.495
C07195=1104.601,364.528,-88.198,-179.703,16.705,151.495
C07196=1104.607,364.775,-88.232,-179.700,16.709,151.496
C07197=1104.613,365.023,-88.268,-179.698,16.712,151.496
C07198=1104.619,365.270,-88.303,-179.694,16.716,151.496
C07199=1104.624,365.517,-88.338,-179.692,16.719,151.497
C07200=1104.630,365.765,-88.374,-179.688,16.723,151.497
C07201=1104.635,366.012,-88.409,-179.686,16.726,151.497
C07202=1104.642,366.259,-88.444,-179.682,16.730,151.497
C07203=1104.647,366.507,-88.479,-179.679,16.734,151.498
C07204=1104.653,366.755,-88.515,-179.677,16.738,151.498
C07205=1104.659,367.002,-88.550,-179.673,16.742,151.498
C07206=1104.664,367.248,-88.585,-179.671,16.745,151.499
C07207=1104.670,367.497,-88.620,-179.668,16.749,151.499
C07208=1104.675,367.744,-88.656,-179.665,16.752,151.499
C07209=1104.681,367.991,-88.691,-179.662,16.756,151.500
C07210=1104.687,368.238,-88.727,-179.660,16.760,151.500
C07211=1104.693,368.486,-88.762,-179.656,16.764,151.500
C07212=1104.698,368.733,-88.798,-179.653,16.768,151.501
C07213=1104.703,368.981,-88.832,-179.651,16.771,151.501
C07214=1104.709,369.228,-88.868,-179.648,16.776,151.502
C07215=1104.718,369.615,-88.924,-179.643,16.781,151.502
C07216=1104.727,370.002,-88.980,-179.639,16.787,151.503
C07217=1104.736,370.388,-89.035,-179.635,16.793,151.503
C07218=1104.745,370.775,-89.091,-179.630,16.799,151.504
C07219=1104.750,371.022,-89.127,-179.627,16.803,151.504
C07220=1104.756,371.270,-89.163,-179.624,16.807,151.505
C07221=1104.762,371.517,-89.198,-179.622,16.811,151.505
C07222=1104.768,371.764,-89.234,-179.619,16.815,151.505
C07223=1104.773,372.011,-89.269,-179.616,16.819,151.506
C07224=1104.779,372.259,-89.305,-179.613,16.823,151.506
C07225=1104.785,372.507,-89.340,-179.610,16.827,151.507
C07226=1104.790,372.754,-89.376,-179.607,16.830,151.507
C07227=1104.796,373.002,-89.412,-179.605,16.835,151.507
C07228=1104.801,373.248,-89.448,-179.601,16.839,151.508
C07229=1104.808,373.496,-89.484,-179.599,16.843,151.508
C07230=1104.813,373.743,-89.519,-179.596,16.847,151.509
C07231=1104.819,373.990,-89.555,-179.593,16.851,151.509
C07232=1104.825,374.238,-89.591,-179.590,16.855,151.509
C07233=1104.831,374.484,-89.627,-179.587,16.859,151.510
C07234=1104.836,374.732,-89.663,-179.585,16.863,151.510
C07235=1104.841,374.979,-89.699,-179.582,16.867,151.511
C07236=1104.848,375.226,-89.735,-179.579,16.871,151.511
C07237=1104.852,375.474,-89.771,-179.576,16.876,151.512
C07238=1104.859,375.721,-89.807,-179.574,16.879,151.512
C07239=1104.865,375.969,-89.842,-179.571,16.884,151.513
C07240=1104.870,376.216,-89.879,-179.568,16.888,151.513
C07241=1104.876,376.463,-89.915,-179.566,16.892,151.514
C07242=1104.881,376.710,-89.951,-179.563,16.896,151.514
C07243=1104.887,376.958,-89.987,-179.560,16.900,151.515
C07244=1104.893,377.205,-90.023,-179.558,16.904,151.515
C07245=1104.898,377.452,-90.059,-179.555,16.909,151.516
C07246=1104.904,377.700,-90.095,-179.552,16.913,151.516
C07247=1104.909,377.946,-90.131,-179.549,16.918,151.517
C07248=1104.915,378.194,-90.167,-179.547,16.922,151.517
C07249=1104.921,378.441,-90.204,-179.544,16.926,151.518
C07250=1104.926,378.688,-90.240,-179.541,16.930,151.518
C07251=1104.932,378.935,-90.277,-179.538,16.935,151.519
C07252=1104.938,379.183,-90.312,-179.536,16.939,151.519
C07253=1104.944,379.429,-90.348,-179.533,16.943,151.520
C07254=1104.949,379.677,-90.385,-179.530,16.948,151.520
C07255=1104.955,379.925,-90.421,-179.527,16.952,151.521
C07256=1104.960,380.171,-90.458,-179.525,16.956,151.521
C07257=1104.966,380.419,-90.494,-179.522,16.961,151.522
C07258=1104.972,380.666,-90.531,-179.519,16.965,151.522
C07259=1104.978,380.913,-90.567,-179.516,16.970,151.523
C07260=1104.983,381.161,-90.603,-179.515,16.974,151.524
C07261=1104.989,381.408,-90.639,-179.512,16.978,151.524
C07262=1104.996,381.655,-90.676,-179.509,16.983,151.525
